METHOD SuperMode : BOOL
VAR_INPUT
END_VAR
IF (*InSync()=TRUE AND *) SyncVertSuperJogExecute_VI AND SuperJogMode_VI THEN
	//jogs are canceled in 'ClearpathLinPPR' FB when SuperJogExecute is set to 0.
	Vert_A.SuperJogExecute_VI :=1;
	Vert_B.SuperJogExecute_VI :=1;
ELSE
	IF JogSeparate_VI = 0 THEN
		Vert_A.SuperJogExecute_VI :=0;
		Vert_B.SuperJogExecute_VI :=0;
	END_IF
END_IF

IF SuperJogMode_VI AND SyncVertSuperJogExecute_VI =0 THEN 	//sync move has to be off to move an individual
	//Vert_A.SuperJogExecute_VI :=VertASuperJog_VI;
	//Vert_B.SuperJogExecute_VI :=VertBSuperJog_VI;

END_IF
END_METHOD

METHOD SyncClampAbsLin : BOOL
VAR_INPUT
END_VAR
IF Clamp_A.Out.InPosition AND Clamp_B.Out.InPosition THEN
	ClampInPosition_PO :=1;
	ELSE ClampInPosition_PO :=0;
END_IF
IF Clamp_A.Out.InTargetPosition AND Clamp_B.Out.InTargetPosition THEN
	ClampInTargetPos_PO :=1;
	else ClampInTargetPos_PO :=0;
END_IF
IF Clamp_A.Out.InMPos AND Clamp_B.Out.InMPos THEN
	ClampIn_M_Pos_PO:=1;
	else ClampIn_M_Pos_PO:=0;
END_IF
CASE SyncClampCase OF
	0: //Ready for move
		IF InSync()=TRUE THEN
			IF Clamp_A.Out.ReadyForMove_PO AND Clamp_B.Out.ReadyForMove_PO THEN
				ClampReadyForMove_PO := TRUE;
				ELSE
					//Msg A or B not readyto move
				END_IF
			ELSE //msg not insync cant move
		END_IF
		IF ClampReadyForMove_PO AND ClampInPosition_PO THEN
			//set request and await execute
			IF bMoveClamp_PI THEN
				Clamp_A.DistancePosReq_PI := ClampDisReq_PI;
				Clamp_B.DistancePosReq_PI := ClampDisReq_PI;
				Clamp_A.bMove_PI :=1;
				Clamp_B.bMove_PI :=1;
				SyncClampCase :=10;
			END_IF
		END_IF
	10: //monitor insync
		bMoveClamp_PI :=0;
		ClampReadyForMove_PO :=FALSE; //step thru case before being able to send again
		IF InSync()=FALSE THEN
			Clamp_A.CancelMove();
			Clamp_B.CancelMove();
			//msg not insync
			SyncClampCase :=90; //syncerror
		END_IF
		//COnfirm Position
		IF ClampInTargetPos_PO THEN
			SyncClampCase:=20;
			ELSE //waiting for move to finish
		END_IF
	20: //Set Ready to Move
		IF InSync()=TRUE THEN
			IF Clamp_A.Out.ReadyForMove_PO AND Clamp_B.Out.ReadyForMove_PO THEN
				ClampReadyForMove_PO := TRUE;
				ELSE
					//Msg A or B not readyto move
				END_IF
			ELSE //msg not insync cant move
		END_IF
		IF ClampReadyForMove_PO THEN SyncClampCase := 0; END_IF
	90: //SyncError
		SyncClampMsg_VO := 'Not in sync abs move was canceld, reset req';
	
END_CASE
END_METHOD

METHOD SyncRotABS : BOOL
VAR_INPUT
END_VAR
IF Rot_A.Out.InPosition AND (Rot_B.Out.InPosition or bFollowerIdleDisengage) THEN
	RotInPosition_PO :=1;
	ELSE RotInPosition_PO :=0;
END_IF
IF Rot_A.Out.InTargetPosition AND (Rot_B.Out.InTargetPosition OR bFollowerIdleDisengage) THEN
	RotInTargetPos_PO :=1;
	ELSE RotInTargetPos_PO :=0;
END_IF
IF Rot_A.Out.InMPos AND Rot_B.Out.InMPos THEN
	RotIn_M_Pos_PO:=1;
	Else RotIn_M_Pos_PO:=0;
END_IF
CASE SyncRotCase OF
	0: //Ready for move
		IF InSync()=TRUE THEN
			IF Rot_A.Out.ReadyForMove_PO AND (Rot_B.Out.ReadyForMove_PO OR bFollowerIdleDisengage) THEN
				RotReadyForMove_PO := TRUE;
				ELSE
					//Msg A or B not readyto move
				END_IF
			ELSE //msg not insync cant move
		END_IF
		IF RotReadyForMove_PO AND RotInPosition_PO THEN
			//set request and await execute
			IF bMoveRot_PI THEN
				Rot_A.DistancePosReq_PI := RotDegReq_PI;
				Rot_B.DistancePosReq_PI := RotDegReq_PI;
				Rot_A.bMove_PI :=1;
				Rot_B.bMove_PI :=1;
				SyncRotCase :=10;
			END_IF
		END_IF
	10: //monitor insync
		bMoveRot_PI :=0;
		RotReadyForMove_PO :=FALSE;	//step thru case before being able to send again
		IF InSync()=FALSE THEN
			Rot_A.CancelMove();
			Rot_B.CancelMove();
			//msg not insync
			SyncRotCase :=90; //syncerror
		END_IF
		//COnfirm Position
		IF RotInTargetPos_PO  THEN
			SyncRotCase:=20;
			ELSE //waiting for move to finish
		END_IF
	20: //Set Ready to Move
		IF InSync()=TRUE THEN
			IF Rot_A.Out.ReadyForMove_PO AND (Rot_B.Out.ReadyForMove_PO or bFollowerIdleDisengage) THEN
				RotReadyForMove_PO := TRUE;
				ELSE
					//Msg A or B not readyto move
				END_IF
			ELSE //msg not insync cant move
		END_IF
		IF RotReadyForMove_PO THEN SyncRotCase := 0; END_IF
	90: //SyncError
		SyncRotMsg_VO := 'Not in sync abs move was canceld, reset req';
	
END_CASE
END_METHOD

METHOD SyncRotJog : BOOL
VAR_INPUT
END_VAR

IF JogSeparate_VI = FALSE THEN
	IF SyncRotJogExecute_VI THEN //JOSEPHBARTONCHANGE IF InSync()=TRUE AND SyncRotJogExecute_VI THEN
		JogRotAExecute_VI :=1;
		JogRotBExecute_VI :=1;
	ELSE
		JogRotAExecute_VI :=0;
		JogRotBExecute_VI :=0;
	END_IF
	ELSE
		//use the jog a or b vi to move items
	
END_IF
END_METHOD

METHOD PUBLIC SyncVertAbsLin : BOOL
VAR_INPUT
END_VAR
IF Vert_A.Out.InPosition AND Vert_B.Out.InPosition THEN
	VertInPosition_PO :=1;
	else VertInPosition_PO :=0;
END_IF
IF Vert_A.Out.InTargetPosition AND Vert_B.Out.InTargetPosition THEN
	VertInTargetPos_PO :=1;
	ELSE VertInTargetPos_PO :=0;
END_IF
IF Vert_A.Out.InMPos AND Vert_B.Out.InMPos THEN
	VertIn_M_Pos_PO :=1;
	ELSE VertIn_M_Pos_PO:=0;
END_IF
CASE SyncVertCase OF
	0: //Ready for move
		IF InSync()=TRUE THEN
			IF Vert_A.Out.ReadyForMove_PO AND Vert_B.Out.ReadyForMove_PO THEN
				VertReadyForMove_PO := TRUE;
				ELSE
					//Msg A or B not readyto move
				END_IF
			ELSE //msg not insync cant move
		END_IF
		IF VertReadyForMove_PO AND VertInPosition_PO THEN
			//set request and await execute
			IF bMoveVert_PI THEN
				Vert_A.DistancePosReq_PI := VertDisReq_PI;
				Vert_B.DistancePosReq_PI := VertDisReq_PI;
				Vert_A.bMove_PI :=1;
				Vert_B.bMove_PI :=1;
				SyncVertCase :=10;
			END_IF
		END_IF
	10: //monitor insync
		bMoveVert_PI :=0;
		VertReadyForMove_PO :=FALSE; //step thru case before being able to send again
		IF InSync()=FALSE THEN
			Vert_A.CancelMove();
			Vert_B.CancelMove();
			//msg not insync
			SyncVertCase :=90; //syncerror
		END_IF
		//Confirm Position
		IF VertInTargetPos_PO THEN
			SyncVertCase:=20;
			ELSE //waiting for move to finish
		END_IF
	20: //Set Ready to Move
		IF InSync()=TRUE THEN
			IF Vert_A.Out.ReadyForMove_PO AND Vert_B.Out.ReadyForMove_PO THEN
				VertReadyForMove_PO := TRUE;
				ELSE
					//Msg A or B not readyto move
				END_IF
			ELSE //msg not insync cant move
		END_IF
		IF VertReadyForMove_PO THEN SyncVertCase := 0; END_IF
	90: //SyncError
		SyncVertMsg_VO := 'Not in sync abs move was canceld, reset req';
	
END_CASE
END_METHOD

METHOD PRIVATE SyncVertJog : BOOL
VAR_INPUT
END_VAR

IF JogSeparate_VI = FALSE THEN
	IF SyncVertJogExecute_VI THEN //IF InSync()=TRUE AND SyncVertJogExecute_VI THEN
		JogVertAExecute_VI :=1;	//JOSEPHBARTONCHANGE1-27-2023 Removed checking in Clamp and Rotary are in synch for vert movement.
		JogVertBExecute_VI :=1;
	ELSE
		JogVertAExecute_VI :=0;
		JogVertBExecute_VI :=0;
	END_IF
	IF InSync()=TRUE AND SyncClampJogExecute_VI THEN
		JogClampAExecute_VI :=1;
		JogClampBExecute_VI :=1;
	ELSE
		JogClampAExecute_VI :=0;
		JogClampBExecute_VI :=0;
	END_IF
	ELSE
		
	//use the jog a or b vi to move items
END_IF
END_METHOD

END_FUNCTION_BLOCK

// ---- Machine System/FBs/CP/ClearpathPositionABS.TcPOU
FUNCTION_BLOCK ClearpathPositionABS //please check comments inside FB to determine clearpath settings before use
VAR_INPUT
	
	//PI (Program Inputs)
		bHomeStart_PI				: BOOL;		//begin Homing sequence
		PowerOn_PI					: BOOL;		//enable motor command from program
		Stop_PI						: BOOL;		//stop command from program
		DistancePosReq_PI			: REAL;		//distanct position request from the program (input in absolute position and valid after homing)
		ManualMove_PI				: BOOL;		//Call manual move method if true
		Mode_PI						: INT;		//0:noMode, 1:Auto, 2:Manual
		bMove_PI					: BOOL;		//begin absolute move 
		VEReq						: LREAL;
		bAltSpeedControl			: BOOL;		//JOSEPHBARTONCHANGE3-28-2023 This allows for outside control of using altspeed
		bPresetMoveTrigger			: BOOL;		//JOSEPHBARTONCHANGE3-28-2023 This allows for tracking when it is a preset position move
		bStopMove			: BOOL;     // Controls the StopMove()
	//VI (visualization input/hmi input)
		HomeReq_VI			: BOOL; 	// Homing sequence
		Reset_VI			: BOOL;		//reset button		
		DisReq_VI			: REAL;		//Disreq for absolute auto move
		JogExecute_VI		: BOOL;		//Call manual move method if true
		SuperJogExecute_VI	: BOOL;		//call super manual move method if true
		SuperJogMode_VI		: bool;		//Super Mode on if true (changes Jog method) use for overtravel or not homed be Cautious
		JogSlow_VI			: BOOL;		//slow manual move
		CW_VI				: BOOL;		//Set Direction for requested move (does not apply to absolute move) True = Clockwise
	//CI (configuration input)
		IN							: CpABS_CI;
		
		EnableOut_FO 		AT %Q* 	: BOOL; 	//enables the clearpath motor
END_VAR
VAR_OUTPUT
	// Outputs
		Out						: CpABS_Out;
		StopCase				: INT; 		//case tracket StopMove()
END_VAR
VAR
	bSimHigh			: BOOL; 	// Simulated High switch for the Rotation axis
	bSimLow				: BOOL; 	// Simulated High switch for the Rotation axis
	AltSpeedCase		: INT;		//case tracker altspeed()
	AltSpeedReq			: BOOL;		//turn altspeed method on
	ResetCase			: int;		//makes a reset instead of an alt speed request (delays the turning off of reset)
	HomeCase			: INT;		//case tracker home()
	JogCase				: INT;		//case tracker Jog()
	SuperJogCase		: INT;		//case tracker SuperJog()
	DisToGoCase			: INT;		//case tracker MoveABSLin() for pulse train que
	PositionCase		: INT;		//case tracker for tracking inposition
	bMoveTrig			: r_trig;	//rtrig for abs move command [used in CNC MDI]
	
	JogReset			: bool;		//used for auto jog reset [stops alt speed from triggering while clearing pulses instead of a full reset]
	SWLimitStatus		: BOOL;		//Used to check if currently within software limits
	error				: INT;		//5: increment error
	PulsesEnabled		: BOOL;		//enable absolute move method to command pulses
	busy				: BOOL;		//move in progress
	MoveComplete		: BOOL;		//all ppr accounted for after move command
	PulseCount			: INT;		//current Pulse Count
	QuePulseDistance	: REAL;		//Distance expected from current pulse train
	expectedPulse		: INT;		//expected pulses from commanded movements at set PPR
	HomeTrig			: R_trig;	//trigger position capture when homing ends
	ATrig				: R_trig;	//counter/trigger to track how many increments of a output have been commanded
	pulseCounter		: r_trig;
	JogRTrig			: R_Trig;	//jog execute trigger
	JogFTrig			: F_Trig;	//Jog Cancel Trigger
	RotRiseLimSwitch		: R_TRIG;	// Rising trigger for rotation limit switch Normally Closed
	RotFallLimSwitch		: F_TRIG;	// Falling trigger for rotation limit switch Normally Open
	ASG					: BOOL;		//all systems go clearpath (if using asg)
	Cancelled			: BOOL;		//move was cancelled requires reset
	CW					: BOOL; 	//direction of motor rotation: CW is true;  CCW is false;
	DistanceToGo		: REAL;		//difference in distance from current position and requested position.  used to determine linear direction
	LastABSEncoder		: DINT;		//last know encoder track to be used for moving status
	isConfigured		: BOOL;		//turns on or off the configuration settings method so it only runs on first scan
	DistPerMRev 		: INT;
	DisPerPulse			: INT;		//distance per pulse based on configuration inputs
	PulsesToSend		: INT;		//Pulses to send for Absolute move
	CWABS				: Bool;		//Direction for abs Move [Check against pulse wrong dir]
	PulseQueSet			: BOOL;		//start pulses for move
	LastDistanceposReq	: REAL;		//last abs move request (keeps track of InTargetPosition)
	ABSHiLimit	: DINT;
	ABSLoLimit 	: Dint;
	//FI (Field Inputs)

	HLFB_FI	 		AT %I*	: BOOL;		// high level feedback sensors
	bInputBCom_FI	AT %I*	: BOOL;		// check sum for inputb signal	(double check that direction is actually signaled to motor)
	ABSEncoder_FI	AT %I*	: DINT;		//absoulte multiturn encoder
	
	//Linear Homing Variables
	bHigh_FI		AT %I*	: BOOL;
	bLow_FI			AT %I*	: BOOL;
	bHome_FI		AT %I*	: BOOL;
	
	bTest : BOOL;
	
	//FO (Field Outputs)
	HLFB24V_FO 			AT %Q*	: BOOL :=1;	//high level feedback 24v power if needed to used el2008 //default set to true so that hlfb is fucntional
	InputAOut_FO 		AT %Q* 	: BOOL; 	//input A of clearpath motor, output from plc
	InputBOut_FO 		AT %Q* 	: BOOL; 	//input B of clearpath motor, output from plc
END_VAR
VAR RETAIN 
	
	
END_VAR

VAR_IN_OUT

END_VAR

(* Check clearpath settings before use*)
	(* Check the input filter setting for inputA and inputB.   Also check PPR setting, CntsPerPulse, HLFBsetting, and The type of axis,  
		Place clearpath in correct mode of operation Mode for this FB is position 
		Check what Homing setting is used on the clearpath motor	
		check to make sure that the resolution of movement commands matches gearbox compatibiltiy, and plc scan compatability
		
		How the FB works Details:
			1st scan sets configuration using MechDrive_CI()
			Each scan CP motor direction is set based off CW variable
			LocatePosition() drives limit switches and rotary cam limit quadrants
			Pulses are counted using ppr() to move with hlfb rising trig counter.  Expected pulses are tracked with inputA_FO rising trig
			Enable checks for enable signal, cancelled state, and stop_PI state before turning on motor or disenable
			reset: cp motors require an enable off to reset after ac loss...ie estop w/contactor.  it also resets cancelled bit and busy bit (requires reset_vi to run)
			
			Moves are called using homing sequence, Absolute movement, or with manual movement and all require homing.
			after homing absolute movement within software limit_CI is available or manual jog.  Manual jog is set to single pulse method by default
			After Homing Position is tracked using 'DistancePos_PO'
			ABsolute move chains clearpath pulses together to create a smooth motion profile. 
				Pulses sent are tracked against 'DistancePosReq_PI' and 'DistancePos_PO'  When expected pulses are within range of requested position then 'pulsecount' is reset
	*)
(*configruation input setting*)
IF isConfigured = 0 THEN MechDrive_CI(); bHigh_FI := TRUE; END_IF	//run once to set configuration on init

//Handle alternate speed
AltSpeedReq := bAltSpeedControl OR AltSpeedReq;
//Pin outs Clockwise (CW) or Counter Clockwise (CCW)
IF CW THEN	InputBOut_FO := 1;	ELSE InputBOut_FO := 0; 	END_IF //sets direction of movement at motor - check this (add bcom direction pin check)
LocatePosition();				//rotary position of the cam wheel  //also includes a double sensor check for SensorCheck_PO  //Also locates position for linear system for limit sensors //Limits
//Triggers
	//pulseCounter(clk:=HLFB_FI);		//high Level feedback counter based off direction (replaced by abs encoder)
	HomeTrig(clk:=Out.Homed_PO);		//used in ppr() to set pulses to zero after homing
	ATrig (clk:=InputAOut_FO);		//counts pulses sent to motor (clearpath should move based on InputA Rising Trig (check settings in CP to be sure - options are for rising or falling trig)
	JogRTrig(CLK:=JogExecute_VI,);	//Starts Jog()
	JogFTrig(CLK:=JogExecute_VI,);	//Cancels Jog() movement
	bMoveTrig(Clk:=bmove_PI,); 		//confirms that move has triggered and then can check MDI MCode Req Pos	
IF Mode_PI = 2 THEN	
	IF SuperJogMode_VI = 0 THEN
		Jog();
	ELSE
		SuperJog();
	END_IF
	out.ModeMsg_VO := 'Manual Mode engaged';
END_IF
IF Mode_PI = 1 THEN
	out.ModeMsg_VO := 'Auto Mode Engaged';
	DistancePosReq_PI:=DisReq_VI;
	MoveAbsLin();
END_IF
	ABSEncoder();			//tracking of the abs encoder against inputB pulses (default for most use cases) use ppr if using the pulse signals from clearpath
	Home();

//moved movedone into movement manual call and abs move call
MoveDone();						//check if movement is complete (will either check pulses against expected pulses or will check for asg
Enable();						//check for motor enable status and try to enable the motor if PowerOn_PI is true
Reset();						//if reset button turn power off, reset cancelled, and reset busy
IF stop_PI THEN CancelMove(); END_IF	//This requires a reset afterwards to move again
IF GVL_HMI.AutoMode THEN StopMove(); END_IF // Must call axis auto stopping every cycle.

METHOD ABSEncoder : BOOL
VAR_INPUT
END_VAR
VAR
	bTest : BOOL;
END_VAR
//pulsecount is now turned into absolute encoder
//will need to check pulsecount math against encoder and confirm rounding does not cause fb and motor to hunt between pulses
Out.DistancePos_PO :=  (ABSEncoder_FI-in.ABSEncoderZero_CI)/in.ABSEncoderScaler_CI;

ABSHiLimit:= (IN.ABSEncoderZero_CI + (In.ABSEncoderScaler_CI*(In.SWLimit_Hi_CI+5))); //JosephBartonChange1-11-2023 THISISIT ABSEncoderZero_CI
ABSLoLimit:= (In.ABSEncoderZero_CI + (IN.ABSEncoderScaler_CI*(In.SWLimit_Lo_CI-5))); //JosephBartonChange1-11-2023
IF ATrig.Q AND Cancelled = 0 THEN //pulse sent counter rtrg
	IF InputBOut_FO = 1 THEN 
		//QuePulseDistance := QuePulseDistance + In.DisPerPulse_CI; //does not account for cnt per rev yet
		PulsesToSend := PulsesToSend-1; //Track ABS Pulses sent  [went pos dir so remove one from que]
		ELSE 
			//QuePulseDistance := QuePulseDistance - In.DisPerPulse_CI;
			PulsesToSend := PulsesToSend+1; //Track ABS Pulses sent  [went neg dir so add one from que]
	END_IF
	//disperpulse_CI must be calibrated on axis and set in settings
END_IF

IF Cancelled = 1 THEN
	//expectedPulse := pulsecount; 			//removed expectedpulse in favor of QuePulseDistance with the abs encoder Ref the linppr if editing
	//QuePulseDistance := 0;
	Out.ExpDistancePos_PO := Out.DistancePos_PO;
END_IF
IF  movecomplete = 1 THEN //ppr mode
	 //Out.ExpDistancePos_PO := PulseCount/2;
	 Out.ExpDistancePos_PO := Out.DistancePos_PO;
	 //QuePulseDistance:=0;
END_IF
IF  PowerOn_PI =0 THEN
	 Out.ExpDistancePos_PO := Out.DistancePos_PO;
	 //QuePulseDistance:=0;
END_IF
Out.DistancePos_PO := Out.DistancePos_PO; //change distancePOs_PO to float if needed
END_METHOD

METHOD PUBLIC AltSpeed : BOOL
VAR_INPUT
END_VAR
(*clearpath requires at least a 20ms delay where the enable signal is pulsed off to realize alternate speed *)

//start
CASE AltSpeedCase OF
	0:
		IF FIND(STR1:='VERT', STR2:=IN.MotorName) = 0 THEN
			altspeedcase := 10;
		ELSE
			altspeedcase := 100;
		END_IF
	10:
		EnableOut_FO := 1;
		AltSpeedCase := 20;
	20:
		EnableOut_FO := 1;
		AltSpeedCase := 30;
	30:
		EnableOut_FO := 0;
		AltSpeedCase := 40;
	40:
		EnableOut_FO := 0;
		AltSpeedCase := 50;
	50:
		EnableOut_FO := 0;
		AltSpeedCase := 60;
	60:	
		EnableOut_FO := 1;
		//Look for 'AltSpeedCase' to be set to '0' in the call function
	
	90: //error or message
	
	100: 
		EnableOut_FO := 1;
		AltSpeedCase := 110;
	110:
		EnableOut_FO := 1;
		AltSpeedCase := 120;
	120:
		EnableOut_FO := 1;
		AltSpeedCase := 130;
	130:
		EnableOut_FO := 0;
		AltSpeedCase := 140;
	140:
		EnableOut_FO := 0;
		AltSpeedCase := 150;
	150:
		EnableOut_FO := 0;
		AltSpeedCase := 200;
	200: 
		EnableOut_FO := 1;
		AltSpeedCase := 110;
	210:
		EnableOut_FO := 1;
		AltSpeedCase := 220;
	220:
		EnableOut_FO := 1;
		AltSpeedCase := 230;
	230:
		EnableOut_FO := 0;
		AltSpeedCase := 240;
	240:
		EnableOut_FO := 0;
		AltSpeedCase := 250;
	250:
		EnableOut_FO := 0;
		AltSpeedCase := 60;
END_CASE
END_METHOD

METHOD PUBLIC CancelMove : BOOL
VAR_INPUT
END_VAR

VAR
	rCanceledEncoderValue : REAL;
END_VAR
EnableOut_FO 	:= 0;		//only way to clear out overstacked increment calls is to turn enable off and then on
//PowerOn_PI		:=0;	//turn off power on [this is a program input and can't be turned off here] check this to see if still needed[was affecting homecase]
Cancelled	:=1;	//cancelled move needs to be reset
Out.ExpDistancePos_PO := Out.DistancePos_PO; //change distancePOs_PO to float if needed
DistancePosReq_PI:=Out.DistancePos_PO;	// get rid of any requestd move during cancel (must recall it after cancel)
DisToGoCase :=0;
PulsesToSend :=0;
//MCODE Flag
AltSpeedReq :=0;	//clear alt speed mode	
AltSpeedCase :=0;	
InputAOut_FO :=0;
// message (move was canceled)
Out.Error4Msg_VO := 'Cancelled, reset to move motor';
END_METHOD

METHOD PUBLIC Enable : BOOL 	//attempts to enable the motor based on stop_PI, Cancelled, and PowerOn_PI
VAR_INPUT
END_VAR
IF Stop_PI =0 AND cancelled =0 AND PowerOn_PI =1 and ResetCase=0 THEN
	EnableOut_FO :=1;
	IF altSpeedReq THEN
		AltSpeed();				//calls altspeed to cycle thru if homing or manual mode requests a slower mode
	END_IF
ELSE 
	EnableOut_FO :=0;	//message to say stop is on (check this)
END_IF


//power on

//check if asg
IF EnableOut_FO =1 AND HLFB_FI =0 THEN
	Out.ErrorMsg_VO := 'Servo enabled but HLFB not on';
END_IF

//if no asg power off and repeat
END_METHOD

METHOD PUBLIC Error : BOOL
VAR_INPUT
END_VAR
// if hlfb pulses do not move in set timeframe after movement call then call error for motor
END_METHOD

METHOD PUBLIC Home : BOOL
VAR_INPUT
END_VAR
//If encoder field is within the CI limits then machine counts as homed.  If homing seq is needed to check slippage periodically it can be added in this method
IF ABSEncoder_FI >= ABSLoLimit AND ABSEncoder_FI <= ABSHiLimit THEN
	out.Homed_PO := 1;
	Out.HomeMsg_VO := 'Axis is within home limits';
	ELSE
		Out.Homed_PO :=0;
		Out.HomeMsg_VO := 'Axis not within home limits check overtravel';
END_IF

//MAIN HOMING SEQUENCE

CASE HomeCase OF 
	0:	//Main home Sequence [Also stops movement]
		
		
		IF HomeReq_VI  THEN	
			IF IN.Limit_NC_NO_CI = 0 THEN	//NC limit switch configuration
				IF bLow_FI THEN //set direction via hmi unless on a limit switch then default to locateposition()
					CW := 0;
					SendPulse();
				ELSE
					CancelMove();
					//in.ABSEncoderZero_CI := ABSEncoder_FI;
					HomeCase :=10;
				END_IF
			ELSE	//NO limit switch configuration
				IF NOT(bLow_FI) THEN //set direction via hmi unless on a limit switch then default to locateposition()
					CW := 0;
					SendPulse();
				ELSE
					CancelMove();
					HomeCase :=10;
				END_IF
			END_IF
			
		ELSE
			IF	Reset_VI  OR Stop_PI THEN		
				CancelMove();
				HomeCase :=10;
			END_IF
		END_IF
	10:	//go for auto jog reset
		IF cancelled THEN HomeCase :=20; END_IF
		
	20: //auto Reset cycle
		IF InLimits(Out.DistancePos_PO) THEN HomeCase :=30; ELSE HomeCase:=95;  END_IF
	30: HomeCase :=31; //10 scan delay
	31: HomeCase :=32;
	32:	HomeCase :=33;
	33: HomeCase :=34;
	34: HomeCase :=35;
	35: HomeCase :=36;
	36: HomeCase :=37;
	37: HomeCase := 38;
	38: HomeCase := 39;
	39: HomeCase :=40;
	40: //send reset
		JogReset := 1;
		HomeCase :=50;
	50: //wait for reset
		IF JogReset=0 THEN HomeCase :=90; END_IF 
	60:
	70:
	80:
	90: IF HomeReq_VI =TRUE THEN HomeCase :=0; END_IF
	95: //outside of limits
		IF Reset_VI THEN HomeCase:=90; END_IF //no autoreset if outside limits
END_CASE
//slippage Test Periodically if desired

//limit switch and home switch configuration
	(*IF IN.HomingSet_CI = 2 THEN //homing sensor not used - home to low sensor
	bHome_FI := bLow_FI; 
	//message homing sensor not used
	END_IF
	
	IF IN.HomingSet_CI = 3 THEN //homing sensor not used - home to Hi sensor
		bHome_FI := bHigh_FI; 
		//message homing sensor not used
	END_IF
	//error catch for if InputBout wire fails and ends up homing unknown direction repeatedly
	IF PowerOn_PI = 0 THEN HomeCase :=0; END_IF
	IF Stop_PI = 1 THEN HomeCase := 0; END_IF
	//check the InputBOut com using EL1008 input channel to determine that the pulse did work
	//message
	IF bhomestart_PI = 1 THEN HomeCase :=0; AltSpeedReq := 1; AltSpeedCase:=0; END_IF
	CASE HomeCase OF
		0://set pulses equal so that movement can begin and check direction
			IF bHomeStart_PI =1 AND Stop_PI = 0  THEN
				HomeCase := 10;
				bhomeStart_PI :=0;
				AltSpeedReq := 1;				//set slow mode and alternate speed in clearpath
				//AltSpeedCase := 0;			//may need this to start slow speed
				//ExpectedPulse := PulseCount;	//Make movement available no matter the pulse count discrepancy
				Out.ExpDistancePos_PO := Out.DistancePos_PO;
				InputAOut_FO :=0;
				Out.Homed_PO :=0;
			END_IF
		(*5:	
			IF Stop_PI = 0  THEN
				HomeCase := 10;
				bhomeStart_PI :=0;
				AltSpeedReq := 1;				//set slow mode and alternate speed in clearpath
				AltSpeedCase := 0;
				ExpectedPulse := PulseCount;	//Make movement available no matter the pulse count discrepancy
				Homed_PO :=0;
			END_IF*)
			
		10:// homing sequence
			IF  Stop_PI = 0  THEN
				Out.Homed_PO :=0;
				//check this: reseting expected to match pulse count so that homeing will start if there is a mismatch
				//decide homing direction and homing method //make flag large enough to hit home switch and the limit switch
				IF IN.Limit_NC_NO_CI =0 THEN	//NC switch configuration
					IF bHigh_FI =1 AND bLow_FI =1 THEN	//using normally closed sensor (flag is not on either limit switch)
						IF IN.HomingSet_CI =2 THEN cw := 0; ELSIF IN.HomingSet_CI =3 THEN cw :=1; END_IF //go to high or low first if no limit switch tripped
					END_IF
				ELSE	//NO switch Configuration
					IF bHigh_FI =0 AND bLow_FI =0 THEN	//using normally closed sensor (flag is not on either limit switch)
						IF IN.HomingSet_CI =2 THEN cw := 0; ELSIF IN.HomingSet_CI =3 THEN cw :=1; END_IF //go to high or low first if no limit switch tripped
					END_IF
				END_IF
				//if inputA is hi then turn off (takes 2 cycles to output an increment at cp motor)
					(*if pulses expected = pulse count then do the next move *)
				IF AltSpeedCase = 60 THEN SendPulse(); END_IF
				IF IN.Limit_NC_NO_CI =0 THEN	//NC switch configuration
					IF bHome_FI =0 THEN //use nc switch for sensor [at home position]
						bHomeStart_PI :=0;
						Cancelmove();
						HomeCase := 20;
					END_IF
					ELSE				//NO switch configuration
					IF bHome_FI =1 THEN //use no switch for sensor [at home position]
					bHomeStart_PI :=0;
					Cancelmove();
					HomeCase := 20;
				END_IF	
				END_IF
				(*check this - add in an extra cycle before setting home that moves away from the 
					homed spot in same direction to confirm trigger positino comes on same side of sensor each time*)
			END_IF
		20:	//extra scan before homed
			HomeCase :=50;	//this scan is required to allow for a cancelled move reset after homing
		
		50://after homing reset motor and cancelled bit
			
				Out.Homed_PO := 1;
				//cancelled :=0;	//resets motor after initial homing
				
				//pulsecount :=0; 
				//expectedPulse :=0;
				Out.DistancePos_PO :=0; //set this to calibrated abs value
				Out.ExpDistancePos_PO :=0; //check this prob need to set to Out.distancepos_po after it calibrates
				testbool := TRUE;
				HomeCase := 0;	//back to the start
		90://reset to default or?
		
	END_CASE *)
END_METHOD

METHOD PUBLIC InLimits : BOOL
VAR_INPUT
	Req	: REAL;	//reqested degree or position from abs move to be evaluated for limits
END_VAR
//only valid after homing
InLimits := TRUE;
IF IN.SWLimit_Hi_CI <=0 OR IN.SWLimit_Lo_CI >0 THEN		//check this (may need to have a neg hi at some point)
	//message to say no limits are set
	Out.Error2Msg_VO := 'No limits are set in CI settings';
	InLimits :=FALSE;	
END_IF
IF Req <= IN.SWLimit_Hi_CI AND Req >= IN.SWLimit_Lo_CI THEN
	InLimits := TRUE;
	ELSE
		InLimits :=FALSE;
		Out.Error2Msg_VO := 'Requested move is outside of software limits';
END_IF
END_METHOD

METHOD PUBLIC Jog : BOOL
VAR_INPUT
END_VAR

//add software limits check this
CASE JogCase OF 
	0:	//Main Jog Sequence [Also stops movement]
		IF JogSlow_VI THEN AltspeedReq :=1; ELSE AltSpeedReq :=0;   END_IF
		
		IF JogExecute_VI AND Out.Homed_PO =1 AND SWLimitStatus=TRUE THEN	//if last move is done then allow for manual increment also required to be at home //check sensor check
			IF IN.Limit_NC_NO_CI = 0 THEN	//NC limit switch configuration
				IF bHigh_FI AND bLow_FI THEN //set direction via hmi unless on a limit switch then default to locateposition()
					IF CW_VI = 1 	THEN	CW := 1; 	ELSE CW:=0; 	END_IF
					IF bhigh_fI = 0	THEN 	CW:=0; 		END_IF
					IF bLow_FI = 0 	THEN 	CW:=1; 		END_IF
				END_IF
			ELSE	//NO limit switch configuration
				IF bHigh_FI =0 AND bLow_FI  = 0 THEN //set direction via hmi unless on a limit switch then default to locateposition()
					IF CW_VI = 1 	THEN	CW := 1; 	ELSE CW:=0; 	END_IF
					IF bhigh_fI = 1	THEN 	CW:=0; 		END_IF
					IF bLow_FI = 1 	THEN 	CW:=1; 		END_IF
				END_IF
			END_IF
			IF AltspeedReq THEN			// slowjog if altspeed is requested and wait for case 60
				IF AltspeedCase = 60 THEN
					SendPulse();
				END_IF
			ELSE
					SendPulse();		//send pulse for reg speed jog
			END_IF
		ELSIF JogExecute_VI THEN
				IF ABSEncoder_FI >= ABSHiLimit OR (IN.Limit_NC_NO_CI = 0 AND bHigh_FI =0) OR (IN.Limit_NC_NO_CI = 1 AND bHigh_FI =1)THEN
					CW := 0;
					SendPulse();		//send pulse for reg speed jog
				ELSIF ABSEncoder_FI <= ABSLoLimit OR (IN.Limit_NC_NO_CI = 0 AND bLow_FI =0) OR (IN.Limit_NC_NO_CI = 1 AND bLow_FI =1) THEN
					CW := 1;					
					SendPulse();		//send pulse for reg speed jog
				END_IF
		ELSE
			IF	JogExecute_VI  = FALSE THEN		
				CancelMove();
				JogCase :=10;
			END_IF
		END_IF
	10:	//go for auto jog reset
		IF cancelled THEN jogCase :=30; END_IF
		
	20: //auto Reset cycle
		IF InLimits(Out.DistancePos_PO) THEN JogCase :=30; ELSE JogCase:=95;  END_IF
	30: JogCase :=31; //10 scan delay
	31: JogCase :=32;
	32:	JogCase :=33;
	33: JogCase :=34;
	34: JogCase :=35;
	35: JogCase :=36;
	36: JogCase :=37;
	37: JogCase := 38;
	38: JogCase := 39;
	39: JogCase :=40;
	40: //send auto jog reset
		JogReset := 1;
		JogCase :=50;
	50: //wait for jog to reset
		IF JogReset=0 THEN JogCase :=90; END_IF 
	60:
	70:
	80:
	90: IF JogExecute_VI =TRUE THEN JogCase :=0; END_IF
	95: //outside of limits
		if Reset_VI then JogCase:=90; End_if //no autoreset if outside limits
	
END_CASE
END_METHOD

METHOD PUBLIC LocatePosition : Bool //determines if sensorcheck is on and working.  Enables movement
VAR_INPUT
END_VAR
	// Setup the switches for rotational axis.
IF IN.bIsRotationAxis THEN
	RotRiseLimSwitch(CLK := bHigh_FI);
	RotFallLimSwitch(CLK := bHigh_FI);
	IF IN.Limit_NC_NO_CI = 0 THEN
		IF RotRiseLimSwitch.Q THEN
			bSimHigh := TRUE;
			bSimLow  := TRUE;
		END_IF
		IF RotFallLimSwitch.Q THEN
			IF CW_VI THEN
				bSimHigh := FALSE;
				bSimLow  := TRUE;
			ELSE
				bSimHigh := TRUE;
				bSimLow  := FALSE;
			END_IF
		END_IF
	ELSE
		IF RotRiseLimSwitch.Q THEN
			bSimHigh := FALSE;
			bSimLow  := FALSE;
		END_IF
		IF RotFallLimSwitch.Q THEN
			IF CW_VI THEN
				bSimHigh := TRUE;
				bSimLow  := FALSE;
			ELSE
				bSimHigh := FALSE;
				bSimLow  := TRUE;
			END_IF
		END_IF
	END_IF
	
	bHigh_FI := bSimHigh;
	bLow_FI  := bSimLow;
END_IF


// Linear axis limit sensors
(*		bHigh_FI		AT %I*	: 	BOOL;
		bLow_FI			AT %I*	: 	BOOL;
		bHome_FI		AT %I*	: 	BOOL;*)
//NC limit sensor configuration
IF IN.Limit_NC_NO_CI = 0 THEN	
	IF bHigh_FI =0 AND bInputBCom_FI =1 AND CW = 1 THEN	//use normally closed sensor and check inputb(-) [applies when trying to move past limit]
		cancelmove();
		CW := 0;	//require next move to be in Neg direction or CCW  //manual move will need to be used to get off limit switch check this
		//message saying that high limit as been exceeded or inputbcom is not connected
		Out.ErrorMsg_VO := 'High Limit reached, reset and move away from limit';
	END_IF
	IF bLow_FI =0 AND bInputBCom_FI = 0 AND CW =0 THEN	//use normally closed sensor and check inputb(-) [applies when trying to move past limit]
		cancelmove();
		CW :=1;	//require next move to be in Neg direction or CCW //manual move will need to be used to get off limit switch check this
		//message saying that Low limit as been exceeded or inputbcom is not connected
		Out.ErrorMsg_VO := 'Low Limit reached, reset and move away from limit';
	END_IF
	//check for abs encoder slip
	IF bHigh_Fi = 0 THEN
		IF ABS(ABSEncoder_FI - ABSHiLimit)> 100 THEN
			Out.Error3Msg_VO := 'Encoder descrepancy at high limit, please confirm no slippage has occured.  Reset encoder calibration in CI settings if needed.';
		END_IF
	END_IF
	IF bLow_FI = 0 THEN
		IF ABS(ABSEncoder_FI - ABSLoLimit)> 100 THEN
			Out.Error3Msg_VO := 'Encoder descrepancy at low limit, please confirm no slippage has occured.  Reset encoder calibration in CI settings if needed.';
		END_IF
	END_IF
ELSE
	//NO limit sensor configuration
	//additional option to use a N/O sensor if desired....not suggested
	IF bHigh_FI =1 AND bInputBCom_FI =1 AND CW = 1 THEN	//use normally closed sensor and check inputb(-) [applies when trying to move past limit]
		cancelmove();
		CW := 0;	//require next move to be in Neg direction or CCW  //manual move will need to be used to get off limit switch check this
		//message saying that high limit as been exceeded or inputbcom is not connected
		Out.ErrorMsg_VO := 'High Limit reached, reset and move away from limit';
	END_IF
	IF bLow_FI =1 AND bInputBCom_FI = 0 AND CW =0 THEN	//use normally closed sensor and check inputb(-) [applies when trying to move past limit]
		cancelmove();
		CW :=1;	//require next move to be in Neg direction or CCW //manual move will need to be used to get off limit switch check this
		//message saying that Low limit as been exceeded or inputbcom is not connected
		Out.ErrorMsg_VO := 'Low Limit reached, reset and move away from limit';
	END_IF
	//check for abs encoder slip
	IF bHigh_Fi = 1 THEN
		IF ABS(ABSEncoder_FI - ABSHiLimit)> 100 THEN
			Out.Error3Msg_VO := 'Encoder descrepancy at high limit, please confirm no slippage has occured.  Reset encoder calibration in CI settings if needed.';
		END_IF
	END_IF
	IF bLow_FI = 1 THEN
		IF ABS(ABSEncoder_FI - ABSLoLimit)> 100 THEN
			Out.Error3Msg_VO := 'Encoder descrepancy at low limit, please confirm no slippage has occured.  Reset encoder calibration in CI settings if needed.';
		END_IF
	END_IF
END_IF
IF Out.DistancePos_PO <=In.SWLimit_Hi_CI AND Out.DistancePos_PO >= In.SWLimit_Lo_CI THEN
	SWLimitStatus := TRUE;
	OUt.LimitsMsg_VO := '';
	ELSE
		SWLimitStatus :=FALSE;
		OUt.LimitsMsg_VO := 'Not inside Software limits, use super mode to move past overtravel';
		//add in ability to jog off of limit
		IF Out.DistancePos_PO >= In.SWLimit_Hi_CI AND CW=1 THEN
			CancelMove();
			CW :=0;
			OUt.LimitsMsg_VO := 'Low SW limit, reset and use super mode to move past overtravel';
		END_IF
		IF Out.DistancePos_PO <= In.SWLimit_Lo_CI AND CW=0 THEN
			CancelMove();
			CW :=1;
			OUt.LimitsMsg_VO := 'High SW limit, reset and use super mode to move past overtravel';
		END_IF
END_IF
END_METHOD

METHOD PUBLIC MechDrive_CI : BOOL
VAR_INPUT
END_VAR
// 0: motor only(rot), 1: Motor and gear(rot), 2: Motor w/gear and screw(lin), 3: Motor w/screw only(lin), 4: Motor w/gear and pulley(lin),  5: Motor w/pulley(lin), 8: bypass mode
(*		DistPerMRev_CI		:	INT;	//distance traveled per rev		(Calculate your own pitch and lead w/gearbox combo must set MechDriveType_CI to 8 to bypass internal calc)
		DegPerMRev_CI		:	INT;	//distance traveled per rev		(Calculate your own pitch and lead w/gearbox combo must set MechDriveType_CI to 8 to bypass internal calc)
		DisPerFPulley_CI	:	INT;	//distance traveled per rev of final pulley (mm)
		GearRatio_CI		:	INT;	// GearRatio motor to moving part (XX:1) (gearbox and lead included in calc for vert axis) (use this for gearbox and pulleys as well)
		Lead_CI				:	INT;	// Lead of Screw if used (mm)			 (gearbox and lead included in calc for vert axis)	
*)

IF IN.MechDriveType_CI = 2 THEN	//2: Motor w/gear and screw(lin)
	DistPerMRev := IN.Lead_CI/IN.GearRatio_CI;	//driven mech ex 4mm/40 = .1mm per rev
	Out.MechTypeMsg_VO := 'Motor w/gear ratio and screw - no Degrees available [no rotary by default]';
	IF IN.GearRatio_CI <=0 OR IN.Lead_CI <=0 THEN
		isconfigured :=0;
		Out.MechTypeMsg_VO := 'GearRatio_CI or Lead_CI not configured please configure to continue';
	END_IF
END_IF

IF IN.MechDriveType_CI = 3 THEN	//3: Motor w/screw only(lin)
	DistPerMRev := IN.Lead_CI;		//driven mech ex 4mm = 4mm per rev
	Out.MechTypeMsg_VO := 'Motor w/screw - no Degrees available [no rotary by default]';
	IF IN.Lead_CI <=0 THEN
		isconfigured :=0;
		Out.MechTypeMsg_VO := 'Lead_CI not configured please configure to continue';
	END_IF
END_IF

IF IN.MechDriveType_CI = 4 THEN	//4: Motor w/gear and pulley(lin),
	DistPerMRev := IN.DisPerFPulley_CI/IN.GearRatio_CI;	//pulley circumference (20t at10 ~ 200mm per fin rev/gear ratio (40) = 5mm/motor rev
	Out.MechTypeMsg_VO := 'Motor w/gear ratio and pulley [no Degree used by default (linear pulley drive) if a rotary either use bypass or use type 1 and include pulley in gear ratio]';
	IF IN.GearRatio_CI <=0 OR IN.DisPerFPulley_CI <=0 THEN
		isconfigured :=0;
		Out.MechTypeMsg_VO := 'GearRatio_CI or DisPerFPulley_CI not configured please configure to continue';
	END_IF
END_IF

IF IN.MechDriveType_CI = 5 THEN	//5: Motor w/pulley(lin);
	DistPerMRev := IN.DisPerFPulley_CI;	//pulley circumference (20t at10 ~ 200mm per fin rev/gear ratio (40) = 5mm/motor rev
	Out.MechTypeMsg_VO := 'Motor w/pulley [no Degree used by default (linear pulley drive) if a rotary either use bypass or use type 1 and include pulley in gear ratio]';
	IF IN.DisPerFPulley_CI <=0 THEN
		isconfigured :=0;
		Out.MechTypeMsg_VO := 'DisPerFPulley_CI not configured please configure to continue';
	END_IF
END_IF

IF IN.MechDriveType_CI = 8 THEN	//8 mechdrivetype is bypassed and is set via DistPerMRev_CI or DegPerMRev_CI;
	DistPerMRev := IN.DistPerMRev_CI;
	Out.MechTypeMsg_VO := 'MechDriveType is bypassed - use DegPerMRev_CI or DistPerMRev_CI';
	IF IN.DistPerMRev_CI <=0  THEN
		isconfigured :=0;
		Out.MechTypeMsg_VO := 'DistPerMRev_CI not configured please configure to continue';
	END_IF
END_IF

IF IN.InputFilter_CI <=0 THEN
	isconfigured :=0;
	Out.ConfigMSG_VO := 'Input filter not configured, please check InputFilter_CI and clearpath motor settings';
END_IF

//linear axis
DisPerPulse := (DistPerMRev*IN.cntpulseSet_CI/32000);	//check this (Likely not a correct calc)
isConfigured :=1;	//sets configuration to true so that this block only runs once
END_METHOD

METHOD PUBLIC MoveAbsLin : BOOL
VAR_INPUT
END_VAR
IF Out.Homed_PO THEN
	CASE PositionCase OF
		0:
			IF ABS(out.DistancePos_PO-LastDistanceposReq) < In.MoveABSTol_CI THEN 
				Out.InTargetPosition:=1; ELSE Out.InTargetPosition:=0; 
			END_IF
			PositionCase :=10;
		10: PositionCase :=20;
		20: PositionCase :=30;
		30: PositionCase :=40;
		40: PositionCase :=50;
		50: PositionCase :=90;
		90: PositionCase :=0;
	END_CASE
	IF ABS(VEReq - Out.DistancePos_PO) < In.MoveABSTol_CI THEN
		Out.InMPos :=1; ELSE Out.InMPos:=0;
	END_IF
	IF bMoveTrig.Q THEN Out.InMPos :=0; END_IF //Set the MPos to false after move command
	CASE DisToGoCase OF
		0:	//Readyto Take Command
			IF ABS(out.DistancePos_PO-Out.ExpDistancePos_PO) < In.MoveABSTol_CI THEN Out.InPosition:=1; END_IF	//check if current pos is within tolerance
			IF Out.InPosition THEN Out.ReadyForMove_PO :=1; END_IF		//Only ready if in position
			IF Out.ReadyForMove_PO THEN
				IF bMove_PI AND InLimits(DistancePosReq_PI)THEN  //If move is within set limits and called in Prog then execute move
					
					DisToGoCase :=10;
					//set MCode Received Bit [Confirm acted in end case] (this is important for aux axis in cnc VE Variable calls)
				END_IF
			END_IF
		10: //check what quePulseDistance should be and set it
			IF bPresetMoveTrigger THEN
				PulsesToSend := REAL_TO_INT((DistancePosReq_PI - Out.DistancePos_PO) * 1.5); //Gets number of pulses to send When moving to set position.
			ELSE
				PulsesToSend := REAL_TO_INT((DistancePosReq_PI - Out.DistancePos_PO)/In.DisPerPulse_CI); //Gets number of pulses to send
			END_IF
			IF PulsesToSend >0 THEN CWABS:=1; ELSE CWABS:=0; END_IF 	//Sets direction for pulses (pos CW[true] neg CW[False]
			bMove_PI :=0;	//Set Req back to false
			LastDistancePosReq := DistancePosReq_PI; //set for target
			Out.ReadyForMove_PO:=0;	//set busy with abs move
			DisToGoCase :=20;
		20: //set the if homed statement for direction control set that here and move to next case
			IF CWABS THEN CW:=1; ELSE CW:=0; END_IF	//Check abs direction each round of pulse send
			IF ABS(PulsesToSend) >0 THEN 
				PulsesEnabled:=1; 
			ELSE 	
				PulsesEnabled :=0;
				DisToGoCase :=30; //if no more pulses move on to case 30 to check the location toleranceS
					// JOSEPHBARTONCHANGE3-28-2023 Reset bPresetMoveTrigger to FALSE, because the move has ended, so no more preset move.
				IF bPresetMoveTrigger THEN
					bPresetMoveTrigger := FALSE;
				END_IF
				
			END_IF	//if any pos or neg pulses then enable pulses
			Out.InPosition :=0;
			IF PulsesEnabled =1 AND Stop_PI = 0 AND EnableOut_FO =1 AND CW = bInputBCom_FI THEN	//check for the motor being on before incrementing the distancepos from disreq	
				//if inputA is hi then turn off (takes 2 cycles to output an increment at cp motor)
				IF CW = CWABS THEN
					SendPulse();	
				ELSE //Message CW Not equal CWABS
						CancelMove();
						Reset_VI := TRUE;
				END_IF	
			ELSE
				error := 5; //check the inputbcom_FI feedback
			END_IF	
			//if input filter of clearpath is too high sometimes these pulses will not register (needed to maintain ability to chain moves)  Otherwise can use asg and movedone
		30: //count pulses and and when enough pulses set pulses(rounded) not enabled set moving tag
			IF ABS(out.DistancePos_PO-DistancePosReq_PI) < In.MoveABSTol_CI THEN
				Out.InPosition:=1; Out.ABSMoveMsg_VO:='In Position';//Position Reached flag and msg
				DisToGoCase := 40;
				ELSE DisToGoCase :=99; //error
			END_IF
			DisToGoCase :=40;
		40: //add a few scan frames to allow inposition and intarget to be bypassed
			DisToGoCase:=41;
		41:	DisToGoCase:=42;
		42:	DisToGoCase:=43;
		43:	DisToGoCase:=44;
		44:	// ready to receive next quedistance
			Out.ReadyForMove_PO :=1;
			//Send MCode confirmation to true
			DisToGoCase:=0;
	END_CASE

END_IF
END_METHOD

METHOD PUBLIC MoveDone : BOOL
VAR_INPUT
END_VAR
//ppr setting of hlfb is required
(*movecomplete is set either when pulsecount lines up exactly or if pulseque is empty and pulsecount is within tolerance*)
	IF Out.DistancePos_PO = Out.ExpDistancePos_PO  THEN	// (check this - add a tolerance here)
		MoveComplete :=1; 
		MoveDone := TRUE;
		busy :=0;			//set busy to zero (these are possibly interchangable until further code added) check this
		ELSE
			MoveDone :=FALSE;
		//is movedone() not completed check this
		//Add in MOVEDONE:=True; check this
	END_IF
	//movecomplete set for absolute move ppr tolerance
END_METHOD

METHOD PUBLIC Reset : BOOL
VAR_INPUT
END_VAR
//delays the turning off of reset so that it sends a full reset instead of an altspeed request
CASE ResetCase OF
	0: 
		(*Original section below for manual reset *)
		IF reset_VI =1 OR JogReset=1 THEN //reset button or auto jog reset [see jog method]
		EnableOut_FO :=0;	//Turn off to reset (power on will finish reset)
		Cancelled :=0;	//reset the cancelled move bit
		busy :=0;	// check this (is reseting busy needed?)
		DisToGoCase:=0;
		bMove_PI:=0;
		ResetCase :=10;
		OUt.MechTypeMsg_VO 		:= '';		
		Out.ConfigMSG_VO		:= '';		
		Out.ErrorMsg_VO			:= '';	
		Out.Error2Msg_VO		:= '';	
		Out.Error3Msg_VO		:='';		
		Out.Error4Msg_VO 		:='';
		Out.HomeMsg_VO 			:='';				
		OUt.LimitsMsg_VO		:='';	
		Out.ABSMoveMsg_VO		:='';
		OUt.SuperJogMsg_VO		:='';
		Out.DisToGoMsg_VO		:='';
		Out.CanceledMsg_VO		:='';
		Out.ModeMsg_VO			:='';
		LastDistanceposReq := Out.DistancePos_PO; //get rid of req diff from curr pos
		END_IF
		(*original section above for manual reset *)
	10: ResetCase:=20;
	20: ResetCase:=30;
	30: ResetCase:=40;
	40: ResetCase:=50;
	50: ResetCase:=60;
	60: ResetCase:=70;
	70: ResetCase:=80;
	80: ResetCase:=90;
	90: 
		ResetCase:=0;
		Reset_Vi:=0;
		JogReset:=0;
	
END_CASE
//reset by turning power off and then on
END_METHOD

METHOD PUBLIC SendPulse : BOOL
VAR_INPUT
END_VAR
//got rid of 'and busy =0'
IF Stop_PI = 0  AND EnableOut_FO =1 AND CW = bInputBCom_FI THEN	//check for the motor being on before incrementing the distancepos from disreq	
	IF InputAOut_FO =1  THEN 
		InputAOut_FO := 0;
	ELSE 
		IF AltSpeedReq THEN
			IF AltspeedCase =60 THEN
				InputAOut_FO :=1;		//else turn true and subtract increment counter
				AltspeedCase :=0;	//reset altspeed
				IF CW =1 THEN Out.ExpDistancePos_PO := Out.ExpDistancePos_PO +1; ELSE Out.ExpDistancePos_PO := Out.ExpDistancePos_PO - 1; END_IF
				//commenting out while testing absencoder
			END_IF
		ELSE
			InputAOut_FO :=1;		//else turn true and subtract increment counter
			IF CW =1 THEN Out.ExpDistancePos_PO := Out.ExpDistancePos_PO +1; ELSE Out.ExpDistancePos_PO := Out.ExpDistancePos_PO - 1; END_IF
			//commenting out while testing absencoder
		END_IF
		MoveComplete :=0;		//set movedone to zero and await move complete
		busy		 :=1;		//set status to busy until move complete
	END_IF	
ELSE
	//InputAOut_FO := 0;		//no trigger if stopped or direction feedback failed or if motor enable is off
	//Message Saying Move is in progress
		
END_IF
END_METHOD

METHOD StopMove : BOOL
VAR_INPUT
END_VAR
(*
	JOSEPHBARTONCHANGE3-23-2023
	This method is to stop motor movement without canceling the entire process.
*)

CASE stopCase OF
	0:
		IF bStopMove THEN
			EnableOut_FO 			:= 0;						//only way to clear out overstacked increment calls is to turn enable off and then on
			Out.ExpDistancePos_PO 	:= Out.DistancePos_PO; 		//change distancePOs_PO to float if needed
			DistancePosReq_PI  		:= Out.DistancePos_PO;		// get rid of any requestd move during cancel (must recall it after cancel)
			DisToGoCase 			:= 0;						// Remove the excess distances
			PulsesToSend 			:= 0;						// Romeve pulses from the pulse buffer
			bMove_PI 				:= 0;						// no move
			AltSpeedReq 			:= FALSE;					// no altspeed
			Out.Error4Msg_VO 		:= 'Motor Move Stopped';	// debugging line to show movement stopped using this function.
			InputAOut_FO := 0;
			MoveComplete := TRUE;
			
			stopCase := stopCase + 10;
		END_IF
		
		
	// Cycle Buffering like jake did.
	// Not sure if you have to do MoveComplete := TRUE every cycle, but Just In Case.
	10: stopCase := stopCase + 10; EnableOut_FO 	:= 0; InputAOut_FO := 0;
	20: stopCase := stopCase + 10; EnableOut_FO 	:= 0; InputAOut_FO := 0;
	30: stopCase := stopCase + 10; EnableOut_FO 	:= 0; InputAOut_FO := 0;
	40: stopCase := stopCase + 10; EnableOut_FO 	:= 0; InputAOut_FO := 0;
	50: stopCase := stopCase + 10; EnableOut_FO 	:= 0; InputAOut_FO := 0;
	60: stopCase := stopCase + 10; EnableOut_FO 	:= 0; InputAOut_FO := 0; 
	70: stopCase := stopCase + 10; EnableOut_FO 	:= 0; InputAOut_FO := 0;
	80: stopCase := stopCase + 10; EnableOut_FO 	:= 0; InputAOut_FO := 0;
	90: stopCase := stopCase + 10; EnableOut_FO 	:= 0; InputAOut_FO := 0;
	
	100: // Reset Case
		MoveComplete := TRUE;
		IF GVL_SAF.DeadmanEnable THEN EnableOut_FO := 1; END_IF		// Re-enable motor to hold motors that are not on a gearbox.
		InputAOut_FO := 0;
		
		IF NOT bStopMove THEN // Reset when ready to not stop.
			stopCase := 0;
		END_IF
		
END_CASE
END_METHOD

METHOD PUBLIC SuperJog : BOOL
VAR_INPUT
END_VAR
//using this mode will disable the two sensor safety check for manual manual mode
//homing is not required to use this and as such should be used with caution
//if not 2 sensors on and not in super mode then no movement allowed
	
	//message : at least one sensor is down please check sensors.  if movement is needed enter supermanual mode
	
//else  allow manual mode  even if not all sensors are working
	//message: you are in supermanual mode and will bypass anti collision devices.  please take caution
//add software limits check this

//add software limits check this
CASE SuperJogCase OF 
	0:	//Main Jog Sequence [Also stops movement]
		IF JogSlow_VI THEN AltspeedReq :=1; ELSE AltSpeedReq :=0;   END_IF
			
		IF SuperJogExecute_VI  THEN	//if last move is done then allow for manual increment also required to be at home //check sensor check
			(*IF IN.Limit_NC_NO_CI = 0 THEN	//NC limit switch configuration
				IF bHigh_FI AND bLow_FI THEN //set direction via hmi unless on a limit switch then default to locateposition()
					IF CW_VI = 1 	THEN	CW := 1; 	ELSE CW:=0; 	END_IF
					IF bhigh_fI = 0	THEN 	CW:=0; 		END_IF
					IF bLow_FI = 0 	THEN 	CW:=1; 		END_IF
				END_IF
				ELSE	//NO limit switch configuration
					IF bHigh_FI =0 AND bLow_FI  = 0 THEN //set direction via hmi unless on a limit switch then default to locateposition()
					IF CW_VI = 1 	THEN	CW := 1; 	ELSE CW:=0; 	END_IF
					IF bhigh_fI = 1	THEN 	CW:=0; 		END_IF
					IF bLow_FI = 1 	THEN 	CW:=1; 		END_IF
				END_IF
			END_IF*)
			IF CW_VI = 1 	THEN	CW := 1; 	ELSE CW:=0; 	END_IF
			IF AltspeedReq THEN			// slowjog if altspeed is requested and wait for case 60
				IF AltspeedCase = 60 THEN
					SendPulse();
					
				END_IF
				ELSE
					SendPulse();		//send pulse for reg speed jog
			END_IF
			ELSE
				IF	SuperJogExecute_VI  = FALSE THEN		
					CancelMove();
					SuperJogCase :=10;
				END_IF
		END_IF
	10:	//
		IF SuperJogExecute_VI =TRUE THEN SuperJogCase :=0; END_IF
		
	
END_CASE
END_METHOD

END_FUNCTION_BLOCK

// ---- Machine System/PRGs/Bogie/WX_CP_Simple.TcPOU
PROGRAM WX_CP_Simple
VAR
	WX1A_Clamp : SimpleClamp;
	WX1B_Clamp : SimpleClamp;
	
	WX2A_Clamp : SimpleClamp;
	WX2B_Clamp : SimpleClamp;
	
	WX3A_Clamp : SimpleClamp;
	WX3B_Clamp : SimpleClamp;
	
	WX4A_Clamp : SimpleClamp;
	WX4B_Clamp : SimpleClamp;
END_VAR

//WX1
WX1B_Clamp(Limit_NC_NO_CI := 0);
WX1A_Clamp(Limit_NC_NO_CI := 0);

//WX2
WX2A_Clamp(Limit_NC_NO_CI := 0);
WX2B_Clamp(Limit_NC_NO_CI := 0);

//WX3
WX3A_Clamp(Limit_NC_NO_CI := 0);
WX3B_Clamp(Limit_NC_NO_CI := 0);

//WX4
WX4A_Clamp(Limit_NC_NO_CI := 0);
WX4B_Clamp(Limit_NC_NO_CI := 0);

END_PROGRAM

// ---- Machine System/FBs/CP/SimpleClamp.TcPOU
FUNCTION_BLOCK SimpleClamp
VAR_INPUT
	ClampRequest : BOOL;
	UnClampRequest : BOOL;
	Limit_NC_NO_CI : BOOL;	// Using NC limit switches =0; Using NO Limit switches =1;
	
END_VAR
VAR_OUTPUT
	
	Clamped : BOOL;
	Unclamped : BOOL;
END_VAR
VAR
	
	//HLFB_FI 			AT %I*	: BOOL;	//high level feedback 
	
	Enable_FO 				AT %Q*  : BOOL;		//Enable ClearPath
	InputAOutCW_FO  		AT %Q* 	: BOOL; 	//input A of clearpath motor, Clockwise request move output from plc
	InputBOutCCW_FO  		AT %Q* 	: BOOL; 	//input B of clearpath motor, CounterClockwise move output from plc
	
	ClampedSensorInput_FI 	AT %I* : BOOL; 
	UnclampedSensorInput_FI AT %I* : BOOL; 
	

	
END_VAR



//Move requests if limit switches are NC

IF Limit_NC_NO_CI = 0 THEN
	IF ClampRequest AND ClampedSensorInput_FI THEN
		Enable_FO := 1;
		InputBOutCCW_FO := 1; //Clamp Direction
	ELSE
		ClampRequest := 0;
	END_IF
	
	IF UnclampRequest AND UnclampedSensorInput_FI THEN
		Enable_FO := 1;
		InputAOutCW_FO := 1; //unClamp Direction
	ELSE
		UnclampRequest :=0;
	END_IF
	
	IF NOT(UnclampRequest) AND NOT(ClampRequest) THEN
		Enable_FO := 0;
		InputAOutCW_FO := 0; //unClamp Direction
		InputBOutCCW_FO := 0; //Clamp Direction
	END_IF
	
	//FB OUTPUTS
	IF NOT(ClampedSensorInput_FI) THEN
		Clamped := 1;
	ELSE
		Clamped := 0;
	END_IF
	
	
	IF NOT(UnclampedSensorInput_FI) THEN
		Unclamped := 1;
	ELSE
		Unclamped := 0;
	END_IF
	
END_IF

END_FUNCTION_BLOCK

// ---- Machine System/PRGs/Bogie/Bogie.TcPOU
PROGRAM Bogie
VAR
	SD1 : sSD;
	SD2 : sSD;
	bTestArms : BOOL; // for testing bogie abs move
	bTest : BOOL;
	SD2_DryCycleEnable : BOOL;
	SD2_DryCycleGCODE_String : STRING;
	SD2_DryCycleOnTrig : R_TRIG;
	CNC_Start_R_Trig  : R_TRIG;
	CNC_Start_TON : TON;
	CNC_Start_TON_COMMAND : BOOL;
	
	fbWX2Handler : FB_AutoMovementHandler;
	
	bBootTest : BOOL := FALSE;
END_VAR
VAR_INPUT

END_VAR
VAR PERSISTENT
	//SD2Per: NC;
END_VAR


RequestNewMolds();

fbWX2Handler(
	WX := ADR(WX_CP.WX2)
);

IF GVL_SAF.EStopOK AND GVL_HMI.AutoMode AND bBootTest THEN
	SD1_Sequence();
	
END_IF
SD1_Control(); //Must be running all of the time
SD2_Control(); //Must be running all of the time

SD1_Status();
SD2_Status();

ACTION RequestNewMolds:
// (Dis)Enable each mold station
//Request Mold in SD1 Load position 1 if done spraying both sides and bogie is out of the spray zone
IF GVL_HMI.WX1Enable AND SD1.bSpray_A_Complete AND SD1.bSpray_B_Complete AND SD1.bInSprayPos = 0 THEN
	
	GVL_CONVEYORS.GL6.BOGIE_REQUEST_LOAD_POS_1 := 1;
	
END_IF

//Request Mold in SD1 Load position 2 if done spraying both sides and bogie is out of the spray zone
IF GVL_HMI.WX2Enable AND SD1.bSpray_A_Complete AND SD1.bSpray_B_Complete AND SD1.bInSprayPos = 0 THEN
	
	GVL_CONVEYORS.GL6.BOGIE_REQUEST_LOAD_POS_2 := 1;
	
END_IF

//Request Mold in SD2 Load position 1 if done spraying both sides and bogie is out of the spray zone
IF GVL_HMI.WX3Enable AND SD2.bSpray_A_Complete AND SD2.bSpray_B_Complete AND SD2.bInSprayPos = 0 THEN
	
	GVL_CONVEYORS.GL8.BOGIE_REQUEST_LOAD_POS_1 := 1;
	
END_IF

//Request Mold in SD2 Load position 2 if done spraying both sides and bogie is out of the spray zone
IF GVL_HMI.WX4Enable AND SD2.bSpray_A_Complete AND SD2.bSpray_B_Complete AND SD2.bInSprayPos = 0 THEN
	
	GVL_CONVEYORS.GL8.BOGIE_REQUEST_LOAD_POS_2 := 1;
	
END_IF
END_ACTION

METHOD SD1_ArmsToLoadOrientation : BOOL;
END_METHOD

ACTION SD1_ArmsToTravelOrientation:
//Rotate the Bogie arms to 90 Degrees for Travel

//WX1 Arms to Travel Pos

//WX2 Arms to Travel Pos
END_ACTION

ACTION SD1_Control:
//SD1 Servo Control 
	SD1.AxisRef();

	CASE SD1.state OF

		INIT_MOVESTATE :	(* initialisation *)
			(* initialize all function blocks *)
			SD1.AxisMoveAbsolute.Execute 	:= FALSE;
			SD1.AxisReset.Execute 			:= FALSE;
			SD1.PosistionRequestAuto 		:= NULL;
				SD1.PosistionRequestManual  := NULL;
			SD1.state := ENABLE_MOVESTATE;
			SD1.AxisStop.Execute := FALSE;

		ENABLE_MOVESTATE :
			IF GVL_SAF.EStopOK THEN
				SD1.AxisPower.Enable := TRUE;
				SD1.AxisPower.Enable_Positive := TRUE;
				SD1.AxisPower.Enable_Negative := TRUE;
				IF SD1.AxisPowerOutputs.Done  THEN
					SD1.state := WAITING_FOR_COMMAND_MOVESTATE;
				ELSIF SD1.AxisPowerOutputs.Error THEN
					SD1.state := ERROR_MOVESTATE;
				END_IF
			END_IF

		WAITING_FOR_COMMAND_MOVESTATE :		(* Wait for Position request *)
			IF GVL_HMI.AutoMode AND SD1.PosistionRequestAuto <> 0 THEN //F_CheckRollerDoor(SD1.AxisReadActualPos.Position,SD1.PosistionRequestAuto,GVL_Doors.FQ3) THEN
				SD1.fTargetPosition := LINT_TO_LREAL(SD1.PosistionRequestAuto);
				SD1.state := NEWTARGETPOSITION_MOVESTATE;
			END_IF
			IF GVL_HMI.ManualMode AND SD1.PosistionRequestManual <> 0 AND GVL_SAF.DeadmanEnable THEN //AND F_CheckRollerDoor(SD1.AxisReadActualPos.Position,SD1.PosistionRequestManual,GVL_Doors.FQ3)THEN
				SD1.fTargetPosition := LINT_TO_LREAL(SD1.PosistionRequestManual);
				SD1.state := NEWTARGETPOSITION_MOVESTATE;
			ELSIF GVL_HMI.ManualMode AND SD1.PosistionRequestManual = 0 AND GVL_SAF.DeadmanEnable THEN //Jogging in manual mode only
				SD1.AxisJog( 
    			Axis			:= SD1.AxisRef,
				JogForward		:= SD1.AxisJog.JogForward,
				JogBackwards	:= SD1.AxisJog.JogBackwards,		
				Mode			:= MC_JOGMODE_CONTINOUS,
				Velocity		:= SD1.fTargetVelocity, 
    			Done			=> SD1.AxisJogOutputs.Done,
    			Busy			=> SD1.AxisJogOutputs.Busy,
    			Active			=> SD1.AxisJogOutputs.Active,
    			CommandAborted	=> SD1.AxisJogOutputs.CommandAborted,
    			Error			=> SD1.AxisJogOutputs.Error,
    			ErrorID			=> SD1.AxisJogOutputs.ErrorID
				);
				IF SD1.AxisStopOutputs.Done THEN
					SD1.state := RESET_MOVESTATE;
				END_IF
			END_IF
			
		NEWTARGETPOSITION_MOVESTATE :		(* move to target position *)
			SD1.AxisMoveAbsolute.Position := SD1.fTargetPosition;		
			SD1.AxisMoveAbsolute.Velocity := SD1.fTargetVelocity;	
			SD1.AxisMoveAbsolute.BufferMode := MC_Buffered;
			SD1.AxisMoveAbsolute.Execute := TRUE;
			IF SD1.AxisMoveAbsoluteOutputs.Done THEN
				SD1.AxisMoveAbsolute.Execute 		:= FALSE;
				//GVL_Doors.FQ2.AutoCloseRequest 		:= 1;
				SD1.PosistionRequestAuto 			:= NULL;
				SD1.PosistionRequestManual  		:= NULL;
				GVL_HMI.SD1_ManualPositionRequest 	:= 0;
				SD1.state := WAITING_FOR_COMMAND_MOVESTATE;
			ELSIF SD1.AxisMoveAbsoluteOutputs.CommandAborted OR SD1.AxisMoveAbsoluteOutputs.Error THEN
				SD1.state := ERROR_MOVESTATE;
			END_IF

		ERROR_MOVESTATE :
			IF SD1.AxisRef.Status.Error THEN
				SD1.state := RESET_MOVESTATE;	(* axis error requires reset *)
			ELSE
				SD1.state := INIT_MOVESTATE;		(* function block errors don't need a reset *)
			END_IF

		RESET_MOVESTATE :
			SD1.AxisReset.Execute := TRUE;
			IF SD1.AxisResetOutputs.Done THEN
				SD1.state := INIT_MOVESTATE;
			ELSIF SD1.AxisResetOutputs.Error THEN
				SD1.state := INIT_MOVESTATE; (* can't do anything here *)
			END_IF
	END_CASE
	
	//Disable drive 
	IF GVL_SAF.EStopOK = 0 OR GVL_HMI.NoMode OR (NOT(GVL_SAF.DeadmanEnable) AND GVL_HMI.ManualMode) THEN
		SD1.AxisPower.Enable := FALSE;
		SD1.state := ERROR_MOVESTATE;
		SD1.PosistionRequestAuto := 0;
		SD1.PosistionRequestManual := 0;
		GVL_HMI.SD1_ManualPositionRequest := 0;
	END_IF
	
	//SD1 Function Block Calls
	SD1.AxisReset(
		Axis 	:= SD1.AxisRef,
		Busy 	=> SD1.AxisResetOutputs.Busy,
		Done 	=> SD1.AxisResetOutputs.Done,
		Error 	=> SD1.AxisResetOutputs.Error,
		ErrorID => SD1.AxisResetOutputs.ErrorID
		);
		
//	SD1.AxisReadActualPos(
//		Axis	:= SD1.AxisRef,
//    	Enable	:= TRUE,
//		//Position=> SD1.AxisReadActualPos.Position,
//		Busy 	=> SD1.AxisReadActualPosOutputs.Busy,
//		Error 	=> SD1.AxisReadActualPosOutputs.Error,
//		ErrorID => SD1.AxisReadActualPosOutputs.ErrorID
//		);

	SD1.AxisPower(
    	Axis		:= SD1.AxisRef,
//		Override	:= SD1.fOverride,
   		Status		=> SD1.AxisPowerOutputs.Done,
    	Busy 		=> SD1.AxisPowerOutputs.Busy,
		Error 		=> SD1.AxisPowerOutputs.Error,
		ErrorID 	=> SD1.AxisPowerOutputs.ErrorID
		);

	SD1.AxisMoveAbsolute(
    	Axis			:= SD1.AxisRef,
    	Done			=> SD1.AxisMoveAbsoluteOutputs.Done,
    	Busy			=> SD1.AxisMoveAbsoluteOutputs.Busy,
    	Active			=> SD1.AxisMoveAbsoluteOutputs.Active,
    	CommandAborted	=> SD1.AxisMoveAbsoluteOutputs.CommandAborted,
    	Error			=> SD1.AxisMoveAbsoluteOutputs.Error,
    	ErrorID			=> SD1.AxisMoveAbsoluteOutputs.ErrorID
		);
	
	SD1.AxisStop(
    	Axis			:= SD1.AxisRef,
		Execute			:= SD1.AxisStop.Execute,
    	Done			=> SD1.AxisStopOutputs.Done,
    	Busy			=> SD1.AxisStopOutputs.Busy,
    	Active			=> SD1.AxisStopOutputs.Active,
    	CommandAborted	=> SD1.AxisStopOutputs.CommandAborted,
    	Error			=> SD1.AxisStopOutputs.Error,
    	ErrorID			=> SD1.AxisStopOutputs.ErrorID
		);
// HMI has problems with handling Enumerations it seems, so HMI Manual buttons are handled here

IF GVL_HMI.SD1_ManualPositionRequest = 1 THEN
	
	SD1.PosistionRequestManual := SprayPos;
	
ELSIF GVL_HMI.SD1_ManualPositionRequest = 2 THEN
 
	SD1.PosistionRequestManual := RollPos;
	
ELSIF GVL_HMI.SD1_ManualPositionRequest = 3 THEN
 
	SD1.PosistionRequestManual := CurePos;
END_IF
END_ACTION

ACTION SD1_Pickup:
IF GVL_HMI.WX1Enable AND SD1.bInSprayPos AND GVL_CONVEYORS.GL6.PP_LOAD_POS_1_IS_ON AND F_PartisPresent(WX1) THEN
	
	//Call pickup of WX1
	
END_IF

IF GVL_HMI.WX2Enable AND SD1.bInSprayPos AND GVL_CONVEYORS.GL6.PP_LOAD_POS_2_IS_ON AND F_PartisPresent(WX2) THEN
	 
	//Call pickup of WX2
	
END_IF
END_ACTION

ACTION SD1_Sequence:
//SD1
IF fbWX2Handler.bError THEN
	SD1.iStep := 900;
END_IF

CASE SD1.iStep OF
	

	0: //Default
		//Do nothing mode. (This means you can't have things that rely on being called EVERY cycle)
		
	10: //Move arms into load position
		fbWX2Handler.nMoveState := Load_Position;
		IF fbWX2Handler.bMoveComplete THEN		
			SD1.iStep := 20;
		END_IF
		
	20: //Drive SD to 'Pickup Position'
		IF SD1.bInPickupPos THEN
			SD1.iStep := 30;
		ELSE
			SD1.PosistionRequestAuto := PickupPos;
		END_IF
	
	30: //Clamp tool
		IF GVL_CONVEYORS.GL6.PP_Load_Pos_1_Is_On AND GVL_HMI.WX1Enable THEN
			//wx1 clamp
		END_IF
		IF GVL_CONVEYORS.GL6.PP_Load_Pos_2_Is_On AND GVL_HMI.WX2Enable THEN
			fbWX2Handler.nMoveState := CLAMP;
		END_IF
		
		IF F_PartIsPresentAndClamped(GVL_IO.WX1) AND F_PartIsPresentAndClamped(GVL_IO.WX2)  THEN 
			SD1.iStep := 40;
		END_IF
		
	40: //Move arms to lifted position
		fbWX2Handler.nMoveState := LIFTED_POSITION;
		IF fbWX2Handler.bMoveComplete THEN
			SD1.iStep := 50;
		END_IF
		
	50: //Jog SD axis to spray position
		IF SD1.bInSprayPos THEN
			SD1.iStep := 70;
		ELSE
			SD1.PosistionRequestAuto := SprayPos;
		END_IF
(*Side A ----------------------------------------------------------------*)		
	60: //Call Side A Spray
		IF PRG_CNCChannelHandler.CNCChannel[0].currentmode = 3 THEN
			PLCMachineMode[0].MDIString := WSTRING_TO_STRING("L C://CNC/TestSpray");
			PLCMachineMode[0].Start := TRUE;
			SD1.bSpray_A_Complete := 0;
		END_IF
		IF SD1.bSpray_A_Complete THEN
			SD1.iStep := 70;
		END_IF
			
	70:	//Move to Roll	
		SD1.PosistionRequestAuto := RollPos;
		IF SD1.bInRollPos THEN 	
			SD1.iStep := 80;
		END_IF
		
	80: //Side A Roll
		IF SD1.bRoll_A_Complete  THEN
			SD1.iStep := 90;
		END_IF
			
	90: //Side A Place Ribs if required It's a database check. From the data in the data structure in the PLC.
		IF SD1.bPlace_A_Complete THEN 
			SD1.iStep := 100;
		END_IF

	100: //Move to Cure
		SD1.PosistionRequestAuto := CurePos;
		IF SD1.bInCurePos THEN
		 	SD1.iStep := 110;
		END_IF	

	110: //Side A Cure
		//Start Heater here 
		IF SD1.bCure_A_Complete THEN
		 	SD1.iStep := 120;
		END_IF
		
(*Side B -----------------------------------------------------------*)
		
	120: //Move to Spray WX Side B & SD
		SD1.PosistionRequestAuto := SprayPos;
		IF SD1.bInSprayPos THEN
			SD1.iStep := 130;
		END_IF
		
	130: //Side B Spray
		IF PRG_CNCChannelHandler.CNCChannel[0].currentmode = 3 THEN
			PLCMachineMode[0].MDIString := WSTRING_TO_STRING("L C://CNC/TestSpray");
			PLCMachineMode[0].Start := TRUE;
			SD1.bSpray_B_Complete := 0;
		END_IF
		IF SD1.bSpray_B_Complete THEN
			SD1.iStep := 135;
		END_IF
			
	135: //Move to Roll
		SD1.PosistionRequestAuto := RollPos;
		IF SD1.bInRollPos THEN 
			SD1.iStep := 140;
		END_IF
		
	140: //Side B Roll
		IF SD1.bRoll_B_Complete  THEN
			SD1.iStep := 150;
		END_IF
			
	150: //Side B Place
		IF SD1.bPlace_B_Complete THEN 
			SD1.iStep := 160;
		END_IF
		
	160: //Move to Cure
		SD1.PosistionRequestAuto := CurePos;
		IF SD1.bInCurePos THEN 
			SD1.iStep := 170;
		END_IF
		
	170: //Side B Cure
		IF SD1.bCure_B_Complete  THEN
			SD1.iStep := 180;
		END_IF
(*
		When the cure is complete, and the putdown zone is not clear, then we need to have a space to keep the arms that is not under the heaters.
			we could over-cure the mold.
			
			For now keep in roll position until the putdown position is clear. (after side B RIB placement)
*)

	(* Move To Putdown & Lifted Position -------------------------------------------------------------------------------------*)
	
	180:	//move to PutDownPos
		IF SD1.bPutDownZoneClear AND fbWX2Handler.nMoveState = STANDBY THEN
			SD1.PosistionRequestAuto := PutDownPos;
			fbWX2Handler.nMoveState := LIFTED_POSITION;
			SD1.iStep := 190;
		END_IF
	190: // Waiting for motor movement completion
		IF SD1.bInPutDownPos AND (NOT fbWX2Handler.nMoveState = LIFTED_POSITION AND fbWX2Handler.bMoveComplete) THEN
			SD1.iStep := 170;
		END_IF
	
	
	(* Arms To Unload Position & Unclamp -------------------------------------------------------------------------------------------*)
		
	170: //Set Down Molds
		IF NOT fbWX2Handler.nMoveState = UNLOAD_POSITION AND NOT fbWX2Handler.bBusy THEN
			fbWX2Handler.nMoveState := UNLOAD_POSITION;
			SD1.iStep := 171;
		END_IF
	171: // Wait for motor movement completion, and then unclamp motor.
		IF NOT fbWX2Handler.nMoveState = UNLOAD_POSITION AND fbWX2Handler.bMoveComplete THEN
			fbWX2Handler.nMoveState := UNCLAMP;
			SD1.iStep := 172;
		END_IF
	172: // Wait for unclamp to finish
		IF NOT fbWX2Handler.nMoveState = UNCLAMP AND fbWX2Handler.bMoveComplete AND NOT fbWX2Handler.bClamped THEN
			SD1.iStep := 180;
		END_IF
		
	(* Backup Traverse, and Arms To Travel Orientation ------------------------------------------------------------------------*)
		
	180: //Move to PostPutDownPos
		SD1.PosistionRequestAuto := PostPutDownPos;
		IF SD1.bInPostPutDownPos AND NOT fbWX2Handler.bClamped THEN
			SD1.iStep := 185; 
		END_IF
		
	185: //Rotate Clamp Arms to Travel Position 90 degrees
		IF NOT fbWX2Handler.bClamped AND SD1.bInPostPutDownPos THEN
			fbWX2Handler.nMoveState := TRAVERSE_POSITION;
			SD1.iStep := 186;
		END_IF
	186: // Waiting for motor movement completion
		IF NOT fbWX2Handler.nMoveState = TRAVERSE_POSITION AND fbWX2Handler.bMoveComplete THEN
			SD1.iStep := 190;
		END_IF
		
	(* Move to start of spray line to pick up next Tool ------------------------------------------------------------------------------------------------*)
	
	190: //Move to Pre Pick up Pos
		IF NOT fbWX2Handler.bBusy THEN 
			SD1.PosistionRequestAuto := PrePickupPos;
		END_IF
		
		IF SD1.bInPrePickupPos THEN 
			SD1.iStep := 3;
		END_IF
		
	(* Errors ------------------------------------------------------------------------------------------------------------------------------------------*)
		
	900: //errors
		IF fbWX2Handler.bError THEN
			SD1.sWXErrorMessage := fbWX2Handler.sErrorMessage;
			SD1.bWXError 		:= TRUE;
		END_IF
		
		IF SD1.bSDError THEN
			SD1.bSDError := TRUE; 
		END_IF
		
END_CASE
END_ACTION

ACTION SD1_SetDown:
IF SD1.bInPutDownPos AND SD1.bPutDownZoneClear AND (GVL_IO.WX1.A.bPP1_Input OR GVL_IO.WX1.A.bPP2_Input OR GVL_IO.WX1.B.bPP1_Input OR GVL_IO.WX1.B.bPP2_Input) THEN
	
	//Call Putdown of WX1
	
END_IF

IF SD1.bInPutDownPos AND SD1.bPutDownZoneClear AND (GVL_IO.WX2.A.bPP1_Input OR GVL_IO.WX2.A.bPP2_Input OR GVL_IO.WX2.B.bPP1_Input OR GVL_IO.WX2.B.bPP2_Input) THEN
	
	//Call Putdown of WX2
	
END_IF
END_ACTION

ACTION SD1_Status:
//Position Window Variables

	SD1.fSprayPosWindowMin		:= SprayPos - SD1.fPosTolerance;
	SD1.fSprayPosWindowMax		:= SprayPos + SD1.fPosTolerance;
	
	SD1.fPrePickupPosWindowMin	:= PrePickupPos - SD1.fPosTolerance;
	SD1.fPrePickupPosWindowMax	:= PrePickupPos + SD1.fPosTolerance;
	
	SD1.fRollPosWindowMin		:= RollPos - SD1.fPosTolerance;
	SD1.fRollPosWindowMax		:= RollPos + SD1.fPosTolerance;

	SD1.fCurePosWindowMin		:= CurePos - SD1.fPosTolerance;
	SD1.fCurePosWindowMax		:= CurePos + SD1.fPosTolerance;

	SD1.fPutDownPosWindowMin 	:= PutDownPos - SD1.fPosTolerance;
	SD1.fPutDownPosWindowMax 	:= PutDownPos + SD1.fPosTolerance;
	
//Position status - check if either in Spray, Roll, or Cure Zone 

	//PREPICKUP POS
	IF SD1.AxisReadActualPos.Position > SD1.fPrePickupPosWindowMin AND
	   SD1.AxisReadActualPos.Position < SD1.fPrePickupPosWindowMax THEN
		SD1.bInPrePickupPos := 1;
	ELSE
		SD1.bInPrePickupPos := 0;
	END_IF
	//SPRAY/PICKUP POS
	IF SD1.AxisReadActualPos.Position > SD1.fSprayPosWindowMin AND
	   SD1.AxisReadActualPos.Position < SD1.fSprayPosWindowMax THEN
		SD1.bInSprayPos := 1;
	ELSE
		SD1.bInSprayPos := 0;
	END_IF
	//ROLL POS
	IF SD1.AxisReadActualPos.Position	> SD1.fRollPosWindowMin AND
	   SD1.AxisReadActualPos.Position < SD1.fRollPosWindowMax THEN
		SD1.bInRollPos := 1;
	ELSE
		SD1.bInRollPos := 0;
	END_IF
	//CURE POS
	IF SD1.AxisReadActualPos.Position > SD1.fCurePosWindowMin AND
	   SD1.AxisReadActualPos.Position < SD1.fCurePosWindowMax THEN
		SD1.bInCurePos := 1;
	ELSE
		SD1.bInCurePos := 0;
	END_IF
	//PUTDOWN POS
	IF SD1.AxisReadActualPos.Position > SD1.fPutDownPosWindowMin AND
	   SD1.AxisReadActualPos.Position < SD1.fPutDownPosWindowMax THEN
		SD1.bInPutDownPos := 1;
	ELSE
		SD1.bInPutDownPos := 0;
	END_IF

//Conveyor Inputs
GVL_IO.WX1.ConveyorLoadPos := GVL_CONVEYORS.GL6.PP_LOAD_POS_1_IS_ON; 
GVL_IO.WX2.ConveyorLoadPos := GVL_CONVEYORS.GL6.PP_LOAD_POS_2_IS_ON; 

//HMI Inputs to Bogie Structure
GVL_IO.WX1.bEnabled := GVL_HMI.WX1Enable;
GVL_IO.WX2.bEnabled := GVL_HMI.WX2Enable;

//Status from CNC
SD1.bSpray_A_Complete 	:= CNCSystem.Channel[0].M[570].bState_rw; 
SD1.bRoll_A_Complete 	:= CNCSystem.Channel[0].M[571].bState_rw;
SD1.bPlace_A_Complete 	:= CNCSystem.Channel[0].M[572].bState_rw;

SD1.bSpray_B_Complete 	:= CNCSystem.Channel[0].M[573].bState_rw; 
SD1.bRoll_B_Complete 	:= CNCSystem.Channel[0].M[574].bState_rw;
SD1.bPlace_B_Complete 	:= CNCSystem.Channel[0].M[575].bState_rw;
END_ACTION

ACTION SD2_ArmsToLoadOrientation:
//Rotate the Bogie arms to 0 Degrees for Picking up part

//WX3 Arms to 0 degrees

//WX4 Arms to 0 degrees
END_ACTION

ACTION SD2_ArmsToTravelOrientation:
//Rotate the Bogie arms to 90 Degrees for Travel

//WX3 Arms to Travel Pos

//WX4 Arms to Travel Pos
END_ACTION

ACTION SD2_Control:
//SD2 Servo Control 
	SD2.AxisRef();

	CASE SD2.state OF

		INIT_MOVESTATE :	(* initialisation *)
			(* initialize all function blocks *)
			SD2.AxisMoveAbsolute.Execute 	:= FALSE;
			SD2.AxisReset.Execute 			:= FALSE;
			SD2.PosistionRequestAuto 		:= NULL;
				SD2.PosistionRequestManual  := NULL;
			SD2.state := ENABLE_MOVESTATE;
			SD2.AxisStop.Execute := FALSE;

		ENABLE_MOVESTATE :
			IF GVL_SAF.EStopOK THEN
				SD2.AxisPower.Enable := TRUE;
				SD2.AxisPower.Enable_Positive := TRUE;
				SD2.AxisPower.Enable_Negative := TRUE;
				IF SD2.AxisPowerOutputs.Done  THEN
					SD2.state := WAITING_FOR_COMMAND_MOVESTATE;
				ELSIF SD2.AxisPowerOutputs.Error THEN
					SD2.state := ERROR_MOVESTATE;
				END_IF
			END_IF

		WAITING_FOR_COMMAND_MOVESTATE :		(* Wait for Position request *)
			IF GVL_HMI.AutoMode AND SD2.PosistionRequestAuto <> 0 THEN //F_CheckRollerDoor(SD2.AxisReadActualPos.Position,SD2.PosistionRequestAuto,GVL_Doors.FQ3) THEN
				SD2.fTargetPosition := LINT_TO_LREAL(SD2.PosistionRequestAuto);
				SD2.state := NEWTARGETPOSITION_MOVESTATE;
			END_IF
			IF GVL_HMI.ManualMode AND SD2.PosistionRequestManual <> 0 AND GVL_SAF.DeadmanEnable THEN //AND F_CheckRollerDoor(SD2.AxisReadActualPos.Position,SD2.PosistionRequestManual,GVL_Doors.FQ3)THEN
				SD2.fTargetPosition := LINT_TO_LREAL(SD2.PosistionRequestManual);
				SD2.state := NEWTARGETPOSITION_MOVESTATE;
			ELSIF GVL_HMI.ManualMode AND SD2.PosistionRequestManual = 0 AND GVL_SAF.DeadmanEnable THEN //Jogging in manual mode only
				SD2.AxisJog( 
    			Axis			:= SD2.AxisRef,
				JogForward		:= SD2.AxisJog.JogForward,
				JogBackwards	:= SD2.AxisJog.JogBackwards,		
				Mode			:= MC_JOGMODE_CONTINOUS,
				Velocity		:= SD2.fTargetVelocity, 
    			Done			=> SD2.AxisJogOutputs.Done,
    			Busy			=> SD2.AxisJogOutputs.Busy,
    			Active			=> SD2.AxisJogOutputs.Active,
    			CommandAborted	=> SD2.AxisJogOutputs.CommandAborted,
    			Error			=> SD2.AxisJogOutputs.Error,
    			ErrorID			=> SD2.AxisJogOutputs.ErrorID
				);
				IF SD2.AxisStopOutputs.Done THEN
					SD2.state := RESET_MOVESTATE;
				END_IF
			END_IF
			
		NEWTARGETPOSITION_MOVESTATE :		(* move to target position *)
			SD2.AxisMoveAbsolute.Position := SD2.fTargetPosition;		
			SD2.AxisMoveAbsolute.Velocity := SD2.fTargetVelocity;	
			SD2.AxisMoveAbsolute.BufferMode := MC_Buffered;
			SD2.AxisMoveAbsolute.Execute := TRUE;
			IF SD2.AxisMoveAbsoluteOutputs.Done THEN
				SD2.AxisMoveAbsolute.Execute 		:= FALSE;
				GVL_Doors.FQ2.AutoCloseRequest 		:= 1;
				SD2.PosistionRequestAuto 			:= NULL;
				SD2.PosistionRequestManual  		:= NULL;
				GVL_HMI.SD2_ManualPositionRequest 	:= 0;
				SD2.state := WAITING_FOR_COMMAND_MOVESTATE;
			ELSIF SD2.AxisMoveAbsoluteOutputs.CommandAborted OR SD2.AxisMoveAbsoluteOutputs.Error THEN
				SD2.state := ERROR_MOVESTATE;
			END_IF

		ERROR_MOVESTATE :
			IF SD2.AxisRef.Status.Error THEN
				SD2.state := RESET_MOVESTATE;	(* axis error requires reset *)
			ELSE
				SD2.state := INIT_MOVESTATE;		(* function block errors don't need a reset *)
			END_IF

		RESET_MOVESTATE :
			SD2.AxisReset.Execute := TRUE;
			IF SD2.AxisResetOutputs.Done THEN
				SD2.state := INIT_MOVESTATE;
			ELSIF SD2.AxisResetOutputs.Error THEN
				SD2.state := INIT_MOVESTATE; (* can't do anything here *)
			END_IF
	END_CASE
	
	//Disable drive 
	IF GVL_SAF.EStopOK = 0 OR GVL_HMI.NoMode OR (NOT(GVL_SAF.DeadmanEnable) AND GVL_HMI.ManualMode) THEN
		SD2.AxisPower.Enable := FALSE;
		SD2.state := ERROR_MOVESTATE;
		SD2.PosistionRequestAuto := 0;
		SD2.PosistionRequestManual := 0;
		GVL_HMI.SD2_ManualPositionRequest := 0;
	END_IF
	
	//SD2 Function Block Calls
	SD2.AxisReset(
		Axis 	:= SD2.AxisRef,
		Busy 	=> SD2.AxisResetOutputs.Busy,
		Done 	=> SD2.AxisResetOutputs.Done,
		Error 	=> SD2.AxisResetOutputs.Error,
		ErrorID => SD2.AxisResetOutputs.ErrorID
		);
		
//	SD2.AxisReadActualPos(
//		Axis	:= SD2.AxisRef,
//    	Enable	:= TRUE,
//		//Position=> SD2.AxisReadActualPos.Position,
//		Busy 	=> SD2.AxisReadActualPosOutputs.Busy,
//		Error 	=> SD2.AxisReadActualPosOutputs.Error,
//		ErrorID => SD2.AxisReadActualPosOutputs.ErrorID
//		);

	SD2.AxisPower(
    	Axis		:= SD2.AxisRef,
//		Override	:= SD2.fOverride,
   		Status		=> SD2.AxisPowerOutputs.Done,
    	Busy 		=> SD2.AxisPowerOutputs.Busy,
		Error 		=> SD2.AxisPowerOutputs.Error,
		ErrorID 	=> SD2.AxisPowerOutputs.ErrorID
		);

	SD2.AxisMoveAbsolute(
    	Axis			:= SD2.AxisRef,
    	Done			=> SD2.AxisMoveAbsoluteOutputs.Done,
    	Busy			=> SD2.AxisMoveAbsoluteOutputs.Busy,
    	Active			=> SD2.AxisMoveAbsoluteOutputs.Active,
    	CommandAborted	=> SD2.AxisMoveAbsoluteOutputs.CommandAborted,
    	Error			=> SD2.AxisMoveAbsoluteOutputs.Error,
    	ErrorID			=> SD2.AxisMoveAbsoluteOutputs.ErrorID
		);
	
	SD2.AxisStop(
    	Axis			:= SD2.AxisRef,
		Execute			:= SD2.AxisStop.Execute,
    	Done			=> SD2.AxisStopOutputs.Done,
    	Busy			=> SD2.AxisStopOutputs.Busy,
    	Active			=> SD2.AxisStopOutputs.Active,
    	CommandAborted	=> SD2.AxisStopOutputs.CommandAborted,
    	Error			=> SD2.AxisStopOutputs.Error,
    	ErrorID			=> SD2.AxisStopOutputs.ErrorID
		);
// HMI has problems with handling Enumerations it seems, so HMI Manual buttons are handled here

IF GVL_HMI.SD2_ManualPositionRequest = 1 THEN
	
	SD2.PosistionRequestManual := SprayPos;
	
ELSIF GVL_HMI.SD2_ManualPositionRequest = 2 THEN
 
	SD2.PosistionRequestManual := RollPos;
	
ELSIF GVL_HMI.SD2_ManualPositionRequest = 3 THEN
 
	SD2.PosistionRequestManual := CurePos;
END_IF
END_ACTION

ACTION SD2_DryCycle:
//SD2

CNC_Start_TON(IN:=CNC_Start_TON_COMMAND,PT:=T#2500MS);

SD2_DryCycleOnTrig(CLK :=SD2_DryCycleEnable);
	IF SD2_DryCycleOnTrig.Q THEN
		SD2.iStepDry := 1;
		
		END_IF
		

IF SD2_DryCycleEnable THEN
	

	Global_HMI.PLCMachineMode[0].MDI := 1;
	Global_HMI.PLCMachineMode[0].ManualMode.nManualTyp := 1;


	CASE SD2.iStepDry OF
//	0: 	//default
	1: SD2.PosistionRequestAuto := SprayPos;
	IF SD2.bInSprayPos 	 THEN 	SD2.iStepDry := 25;	END_IF
    5:	//Check that WX1 and WX2 are empty and do not contain a mold, then rotate arms to Load Orientation
		IF SD2.bInPrePickupPos THEN
			SD2_ArmsToLoadOrientation();
		END_IF
		SD2.iStepDry := 10;
	10: //Move to Spray/Pickup Pos
		IF SD2.bInPrePickupPos THEN
			SD2.PosistionRequestAuto := SprayPos;				
		END_IF
		IF SD2.bInSprayPos 	 THEN 	SD2.iStepDry := 15;	END_IF
	15: //Check if there there molds ready for pickup and pickup if mold present and WX is enabled
		IF SD2.bInSprayPos THEN SD2.iStepDry := 25; END_IF
//	17: 
//		CNC_Start_TON_COMMAND := 1;
//		SD2.iStepDry := 20;
		
//	20: //Side A Spray

//		IF PRG_CNCChannelHandler.CNCChannel[0].currentmode = 3 THEN
//			PLCMachineMode[0].MDIString := 'G01 X1700 F9000 
//G01 Y4000 F5000
//G01 X1400 F9000
//G01 Y2000 F5000';
			

//			IF CNC_Start_TON.ET < T#2500MS AND CNC_Start_TON.ET > T#0MS THEN
//				PLCMachineMode[0].Start := TRUE;
//			END_IF
//			IF CNC_Start_TON.Q THEN
//				CNC_Start_TON_COMMAND := 0;
//				PLCMachineMode[0].Start := FALSE;
			
//			END_IF
		
//		END_IF
		
//		IF Global_HMI.PLCMachineMode[0].Ready = 1 THEN	SD2.iStepDry := 25;	END_IF
	25:	//Move to Roll	
		SD2.PosistionRequestAuto := RollPos;
		IF SD2.bInRollPos  THEN 	SD2.iStepDry := 190;	END_IF
	190: //Move to Pre Pick up Pos
		
		SD2.PosistionRequestAuto := PrePickupPos;
		
		IF SD2.bInPrePickupPos THEN SD2.iStepDry := 5; END_IF
	END_CASE
END_IF
END_ACTION

ACTION SD2_Pickup:
IF GVL_HMI.WX3Enable AND SD1.bInSprayPos AND GVL_CONVEYORS.GL6.PP_LOAD_POS_1_IS_ON AND F_PartisPresent(WX3) THEN
	
	//Call pickup of WX3
	
END_IF

IF GVL_HMI.WX4Enable AND SD1.bInSprayPos AND GVL_CONVEYORS.GL6.PP_LOAD_POS_2_IS_ON AND F_PartisPresent(WX4) THEN
	 
	//Call pickup of WX4
	
END_IF
END_ACTION

ACTION SD2_Sequence:
//SD2
	(* seq begins when 2 molds are picked up.  Their GCode file 'strings' should be stored in RFID Tag *)
	//Call PickupSD2()
	//Add Mold Job Files to Spray Que [FIFO] 
		//WX1:Key_A, WX1:Macro_A, WX2:Key_A, WX2:Macro_A, WX1:Key_B, WX1:Macro_B, WX2:Key_B, WX2:Macro_B
	//Add Mold Job Files to Roll Que [FIFO]
		//WX1:Key_A, WX1:Macro_A, WX2:Key_A, WX2:Macro_A, SoftCureSideA, WX1:Key_B, WX1:Macro_B, WX2:Key_B, WX2:Macro_B, SOFTCureSideB
	//Add Mold Job Files to Place Que [FIFO] (*These will prob need a FIFO Priority but allow for opportunity running on SD2*)
		//WX1:Side_A, WX2:Side_A, WX1:Side_B, WX2:Side_B 
	//Await Job Complete then --- Call SetDownSD2()
	//SD2 Case
	CASE SD2.iStep OF
	0: 	//default
	5:	//Check that WX1 and WX2 are empty and do not contain a mold, then rotate arms to Load Orientation
		IF F_IsEmpty(WX1) = 0 AND F_IsEmpty(WX2) AND SD2.bInPrePickupPos THEN
			SD2_ArmsToLoadOrientation();
		END_IF
		SD2.iStep := 10;
	10: //Move to Spray/Pickup Pos
		IF SD2.bInPrePickupPos AND F_ArmsInLoadOrientation() THEN
			SD2.PosistionRequestAuto := SprayPos;				
		END_IF
		IF SD2.bInSprayPos 		 THEN 	SD2.iStep := 15;	END_IF
	15: //Check if there there molds ready for pickup and pickup if mold present and WX is enabled
		IF SD2.bInSprayPos THEN SD2_Pickup(); END_IF
	
		IF F_PartPickupSuccess(WX1) AND F_PartPickupSuccess(WX2) THEN
			SD2.iStep := 17;
			ELSE
			SD2.iStep := 0;
			//No Mold to pick up 
		END_IF
	17: //Add Files to Que
		IF F_PartIsPresent(WX1) THEN
			//Get mold id and Database data and put into WX1.CurrentJob
			//Load files for WX1 
			WX1.CurrentJob.AKeyFile := 'test.nc';
		END_IF
		IF F_PartIsPresent(WX2) THEN
			//Load files for WX2
			WX2.CurrentJob.AKeyFile := 'test2.nc';
			//Get mold id and Database data and put into WX2.CurrentJob
		END_IF
		//check if files present and loaded
		IF F_CheckMoldData(WX1.CurrentJob.MoldID,GVL_HMI.WX1Enable) AND F_CheckMoldData(WX1.CurrentJob.MoldID,GVL_HMI.WX1Enable) THEN
			SD2.iStep := 20;
			ELSE
				//Mold Data missing or incorrect
		END_IF
	20: //Side A Spray
		IF SD2.bSpray_A_Complete THEN	SD2.iStep := 25;	END_IF
	25:	//Move to Roll	
		SD2.PosistionRequestAuto := RollPos;
		IF SD2.bInRollPos 		 THEN 	SD2.iStep := 30;	END_IF
	30: //Side A Roll
		IF SD2.bRoll_A_Complete  THEN	SD2.iStep := 40;	END_IF
	40: //Side A Place
		IF SD2.bPlace_A_Complete THEN 	SD2.iStep := 45;	END_IF
	45: //Move to Cure
		SD2.PosistionRequestAuto := CurePos;
		IF SD2.bInCurePos 		 THEN 	SD2.iStep := 50;	END_IF
	50: //Side A Cure
		IF SD2.bCure_A_Complete  THEN 	SD2.iStep := 55;	END_IF
	55: //Move to Spray
		SD2.PosistionRequestAuto := SprayPos;
		IF SD2.bInSprayPos 		 THEN 	SD2.iStep := 120;	END_IF
	120: //Side B Spray
		IF SD2.bSpray_B_Complete THEN	SD2.iStep := 125;	END_IF
	125: //Move to Roll
		SD2.PosistionRequestAuto := RollPos;
		IF SD2.bInRollPos 		 THEN 	SD2.iStep := 130;	END_IF
	130: //Side B Roll
		IF SD2.bRoll_B_Complete  THEN	SD2.iStep := 140;	END_IF
	140: //Side B Place
		IF SD2.bPlace_B_Complete THEN 	SD2.iStep := 145;	END_IF
	145: //Move to Cure
		SD2.PosistionRequestAuto := CurePos;
		IF SD2.bInCurePos 		 THEN 	SD2.iStep := 150;	END_IF
	150: //Side B Cure
		IF SD2.bCure_B_Complete  THEN	SD2.iStep := 165;	END_IF
	165:	//move to PutDownPos
		IF SD2.bPutDownZoneClear THEN
			SD2.PosistionRequestAuto := PutDownPos;
		END_IF
		IF SD2.bInPutDownPos 	 THEN 	SD2.iStep := 170;	END_IF
	170: //Set Down Molds
		IF SD2.bJob_Complete	THEN
			SD2_SetDown(); 
		END_IF
	180: //Move to PostPutDownPos
		IF WX1.A.bClampLimitLow AND WX1.B.bClampLimitLow AND 
		   WX2.A.bClampLimitLow AND WX2.B.bClampLimitLow THEN
			SD2.PosistionRequestAuto := PostPutDownPos;
		END_IF
		IF SD2.bInPostPutDownPos AND F_IsEmpty(WX1) AND F_IsEmpty(WX2)  THEN SD2.iStep := 185; END_IF
	185: //Rotate Clamp Arms to Travel Position 90 degrees
		SD2_ArmsToTravelOrientation();
		IF WX1.bArmsAtTravelPos AND WX2.bArmsAtTravelPos THEN SD2.iStep := 190;	END_IF
	190: //Move to Pre Pick up Pos
		IF WX1.bArmsAtTravelPos AND WX2.bArmsAtTravelPos THEN 
			SD2.PosistionRequestAuto := PrePickupPos;
			ELSE
				SD2_ArmsToTravelOrientation();
		END_IF
		
		IF SD2.bInPrePickupPos THEN SD2.iStep := 5; END_IF
	900: //errors
	END_CASE
END_ACTION

ACTION SD2_SetDown:
IF SD2.bInPutDownPos AND SD2.bPutDownZoneClear AND (GVL_IO.WX3.A.bPP1_Input OR GVL_IO.WX3.A.bPP2_Input OR GVL_IO.WX3.B.bPP1_Input OR GVL_IO.WX3.B.bPP2_Input) THEN
	
	//Call Putdown of WX3
	
END_IF

IF SD2.bInPutDownPos AND SD2.bPutDownZoneClear AND (GVL_IO.WX4.A.bPP1_Input OR GVL_IO.WX4.A.bPP2_Input OR GVL_IO.WX4.B.bPP1_Input OR GVL_IO.WX4.B.bPP2_Input) THEN
	
	//Call Putdown of WX4
	
END_IF
END_ACTION

ACTION SD2_Status:
//Position Window Variables

	SD2.fSprayPosWindowMin		:= SprayPos - SD2.fPosTolerance;
	SD2.fSprayPosWindowMax		:= SprayPos + SD2.fPosTolerance;
	
	SD2.fPrePickupPosWindowMin	:= PrePickupPos - SD2.fPosTolerance;
	SD2.fPrePickupPosWindowMax	:= PrePickupPos + SD2.fPosTolerance;
	
	SD2.fRollPosWindowMin		:= RollPos - SD2.fPosTolerance;
	SD2.fRollPosWindowMax		:= RollPos + SD2.fPosTolerance;
	
	SD2.fCurePosWindowMin		:= CurePos - SD2.fPosTolerance;
	SD2.fCurePosWindowMax		:= CurePos + SD2.fPosTolerance;

	SD2.fPutDownPosWindowMin 	:= PutDownPos - SD2.fPosTolerance;
	SD2.fPutDownPosWindowMax 	:= PutDownPos + SD2.fPosTolerance;
	
//Position status - check if either in Spray, Roll, or Cure Zone 

	//PREPICKUP POS
	IF SD2.AxisReadActualPos.Position > SD2.fPrePickupPosWindowMin AND
	   SD2.AxisReadActualPos.Position < SD2.fPrePickupPosWindowMax THEN
		SD2.bInPrePickupPos := 1;
	ELSE
		SD2.bInPrePickupPos := 0;
	END_IF
	//SPRAY/PICKUP POS
	IF SD2.AxisReadActualPos.Position > SD2.fSprayPosWindowMin AND
	   SD2.AxisReadActualPos.Position < SD2.fSprayPosWindowMax THEN
		SD2.bInSprayPos := 1;
	ELSE
		SD2.bInSprayPos := 0;
	END_IF
	//ROLL POS
	IF SD2.AxisReadActualPos.Position	> SD2.fRollPosWindowMin AND
	   SD2.AxisReadActualPos.Position < SD2.fRollPosWindowMax THEN
		SD2.bInRollPos := 1;
	ELSE
		SD2.bInRollPos := 0;
	END_IF
	//CURE POS
	IF SD2.AxisReadActualPos.Position > SD2.fCurePosWindowMin AND
	   SD2.AxisReadActualPos.Position < SD2.fCurePosWindowMax THEN
		SD2.bInCurePos := 1;
	ELSE
		SD2.bInCurePos := 0;
	END_IF
	//PUTDOWN POS
	IF SD2.AxisReadActualPos.Position > SD2.fPutDownPosWindowMin AND
	   SD2.AxisReadActualPos.Position < SD2.fPutDownPosWindowMax THEN
		SD2.bInPutDownPos := 1;
	ELSE
		SD2.bInPutDownPos := 0;
	END_IF

//Conveyor Inputs
GVL_IO.WX3.ConveyorLoadPos := GVL_CONVEYORS.GL6.PP_LOAD_POS_1_IS_ON; //JosephBartonChange1-11-2023 I made these both the proper WX3&4 instead of 1&2
GVL_IO.WX4.ConveyorLoadPos := GVL_CONVEYORS.GL6.PP_LOAD_POS_2_IS_ON; //JosephBartonChange1-11-2023 

//HMI Inputs to Bogie Structure
GVL_IO.WX3.bEnabled := GVL_HMI.WX3Enable; //JosephBartonChange1-11-2023 I also made these the proper WX3&4 instead of 1&2
GVL_IO.WX4.bEnabled := GVL_HMI.WX4Enable; //JosephBartonChange1-11-2023
END_ACTION

END_PROGRAM

// ---- Machine System/FBs/FB_AutoMovementHandler.TcPOU
FUNCTION_BLOCK FB_AutoMovementHandler
VAR_INPUT
	// Bogie arms to use
	WX : POINTER TO BogieComboWX;
	
	// State Handler case
	nMoveState : eBogieHandlerCase := STANDBY;
END_VAR
	
VAR_OUTPUT
	//Status Variables
	bMoveComplete : BOOL 		:= FALSE;
	bBusy 		  : BOOL 		:= FALSE; // While bBusy := TRUE; assume motor movement.
	bClamped	  : BOOL 		:= FALSE;
	bHomed    	  : BOOL		:= FALSE;
	
	// Error Variables
	bError 		  : BOOL 		:= FALSE;
	sErrorMessage : STRING(255) := '';
	
	bTest : BOOL;
END_VAR

VAR
	// Bogie arm target position
	WX2TargetPos : sBogieArmPosition;
	
	//Clamp Error Detection
	nWX2ClampedAPos	: LREAL;
	nWX2ClampedBPos : LREAL;
	nClampTolerance : INT := 2;
	
	//Timeout Error Detection
	tStartTime : TIME;
	tTimeLimit : TIME := T#45S;
	
	// General Vars
	nCounter : USINT := 0;
	
	//Initialising Variables
	bInit 	 : BOOL := FALSE;
	
	//Motor Movement Variables
	bCleanUp 			: BOOL := FALSE;
	bCleanUpBusy		: BOOL := FALSE;
	bInitCleanUpTrigger : BOOL := FALSE;
	
	//Clamping Variables
	nClamp_ATracker : ARRAY[1..100] OF REAL;
	nClamp_BTracker : ARRAY[1..100] OF REAL;
		
	nClampAvgPos	: REAL;
	nClampCounter : INT := 1;	// Don't use me.
	
	bClamp_AClamped : BOOL := FALSE;
	bClamp_BClamped : BOOL := FALSE;
	
	bAllStop : BOOL;
	
	// For stopping movement & changing modes
	nStopCounter : INT := 0;	// Don't use me.
END_VAR

VAR CONSTANT
	WX2TravelPos 	: sBogieArmPosition := (
						nVertPos 	   := 0,
						nVertTolerance := 5,
						
						nRotPos := -300,
						nRotTolerance := 5,
						
						nClampPos := 15,
						nClampTolerance := 2
						);
						
	WX2LoadPos 	: sBogieArmPosition := (
						nVertPos 	   := 0,
						nVertTolerance := 5,
						
						nRotPos := 0,
						nRotTolerance := 5,
						
						nClampPos := 15,
						nClampTolerance := 2
						);
	WX2UnloadPos 	: sBogieArmPosition := (
						nVertPos 	   := 0,
						nVertTolerance := 5,
						
						nRotPos := 0,
						nRotTolerance := 5,
						
						nClampPos := 15,
						nClampTolerance := 2
						);
	WX2SprayAPos 	: sBogieArmPosition := (
						nVertPos 	   := 200,
						nVertTolerance := 5,
						
						nRotPos := -300,
						nRotTolerance := 5,
						
						nClampPos := 450,
						nClampTolerance := 2
						);
						
	WX2SprayBPos 	: sBogieArmPosition := (
						nVertPos 	   := 200,
						nVertTolerance := 5,
						
						nRotPos := 300,
						nRotTolerance := 5,
						
						nClampPos := 450,
						nClampTolerance := 2
						);
						
	WX2LiftedPos 	: sBogieArmPosition := (
						nVertPos 	   := 200,
						nVertTolerance := 5,
						
						nRotPos := 0,
						nRotTolerance := 5,
						
						nClampPos := 450,
						nClampTolerance := 2
						);
END_VAR

IF WX^.bPresetMoveTrigger THEN
	WX^.bPresetMoveTrigger := FALSE;
END_IF

bAllStop := allAxisAreStopped();

IF bError AND NOT nMoveState = REMOVE_ERROR THEN
	nMoveState := ERROR;
END_IF

IF bCleanUp THEN
	enableAltSpeed();
END_IF

 // WX1^.Vert_A.Out.DistancePos_PO; To get the current location.
IF NOT bInit THEN
	bInit := TRUE;
END_IF

IF GVL_HMI.AutoMode THEN
	CASE nMoveState OF
		STANDBY: // Do Nothing
			IF bBusy AND NOT bError THEN
				nMoveState := STOP_EXTENDED;
				stopAllMovement();
				disableAltSpeed();
				nCounter := 0;
			END_IF
			
			IF bError THEN nMoveState := ERROR; END_IF
			
		LOAD_POSITION: // Load Position -------------------------------------------------------
			
			IF NOT bBusy THEN
				bBusy := TRUE;
				bMoveComplete := FALSE;
				
				WX2TargetPos := WX2LoadPos;

				WX^.VertDisReq_PI 	:= REAL_TO_INT(WX2TargetPos.nVertPos);
				WX^.RotDegReq_PI  	:= REAL_TO_INT(WX2TargetPos.nRotPos);
				WX^.ClampDisReq_PI := 3; // We can assume we are unclamped.
				
				WX^.Clamp_A.bStopMove := FALSE;
				WX^.Clamp_B.bStopMove := FALSE;
				
				startAllMovement();
				
				disableAltSpeed();
				WX^.bPresetMoveTrigger := TRUE;
				
				nMoveState := MAIN_MOVE;
				
				tStartTime := TIME();
				
			ELSE
				nMoveState := STOP;
			END_IF
			
		TRAVERSE_POSITION: // Goto traverse Position -------------------------------------------------------
			
			IF NOT bBusy THEN
				bBusy := TRUE;
				bMoveComplete := FALSE;
				
				WX2TargetPos := WX2TravelPos;

				WX^.VertDisReq_PI 	:= REAL_TO_INT(WX2TargetPos.nVertPos);
				WX^.RotDegReq_PI  	:= REAL_TO_INT(WX2TargetPos.nRotPos);
				WX^.ClampDisReq_PI := REAL_TO_INT(WX^.Clamp_A.Out.DistancePos_PO); // We can assume we are unclamped.
				
				startAllMovement();
				
				disableAltSpeed();
				WX^.bPresetMoveTrigger := TRUE;
				
				nMoveState := MAIN_MOVE;
				
				tStartTime := TIME();
				
			ELSE
				nMoveState := STOP;
			END_IF

		SPRAY_POSITION_A: // Spray Side A -------------------------------------------------------
			IF NOT bBusy THEN
				bBusy := TRUE;
				bMoveComplete := FALSE;
				
				WX2TargetPos := WX2SprayAPos;
				
				WX^.VertDisReq_PI 	:= REAL_TO_INT(WX2TargetPos.nVertPos);
				WX^.RotDegReq_PI  	:= REAL_TO_INT(WX2TargetPos.nRotPos);
				
				WX2TargetPos.nClampPos := WX^.Clamp_A.Out.DistancePos_PO;
				
				startAllMovement();
				disableAltSpeed();
				WX^.bPresetMoveTrigger := TRUE;
				
				nMoveState := MAIN_MOVE;
				
				tStartTime := TIME();
			END_IF
			
		SPRAY_POSITION_B: // Spray Side B -----------------------------------------------------
			IF NOT bBusy THEN
				bBusy := TRUE;
				bMoveComplete := FALSE;
				
				WX2TargetPos := WX2SprayBPos;
				
				WX^.VertDisReq_PI 	:= REAL_TO_INT(WX2TargetPos.nVertPos);
				WX^.RotDegReq_PI  	:= REAL_TO_INT(WX2TargetPos.nRotPos);
				WX2TargetPos.nClampPos := WX^.Clamp_A.Out.DistancePos_PO;
				
				startAllMovement();
				disableAltSpeed();
				WX^.bPresetMoveTrigger := TRUE;
				
				nMoveState := MAIN_MOVE;
				
				tStartTime := TIME();
			END_IF
		
		UNLOAD_POSITION: // Unload Position ||| THIS NEEDS TO BE CHECKED!
			IF NOT bBusy THEN
				bBusy := TRUE;
				bMoveComplete := FALSE;
				
				WX2TargetPos := WX2UnloadPos;
				
				WX^.VertDisReq_PI 	:= REAL_TO_INT(WX2TargetPos.nVertPos);
				WX^.RotDegReq_PI  	:= REAL_TO_INT(WX2TargetPos.nRotPos);
				WX^.ClampDisReq_PI := REAL_TO_INT(WX2TargetPos.nClampPos);
				
				startAllMovement();
				disableAltSpeed();
				WX^.bPresetMoveTrigger := TRUE;
				
				nMoveState := MAIN_MOVE;
				
				tStartTime := TIME();
			END_IF
		
		LIFTED_POSITION:	
			IF NOT bBusy THEN
				bBusy := TRUE;
				bMoveComplete := FALSE;
				
				WX2TargetPos := WX2LiftedPos;
				
				WX^.VertDisReq_PI 	:= REAL_TO_INT(WX2TargetPos.nVertPos);
				WX^.RotDegReq_PI  	:= REAL_TO_INT(WX2TargetPos.nRotPos);
				WX^.ClampDisReq_PI := REAL_TO_INT(WX2TargetPos.nClampPos);
				
				startAllMovement();
				disableAltSpeed();
				WX^.bPresetMoveTrigger := TRUE;
				
				nMoveState := MAIN_MOVE;
				
				tStartTime := TIME();
			END_IF
			
		CLAMP: // Clamp Tool ||||| THIS NEEDS TO BE CHECKED!
			IF NOT bBusy THEN
				bBusy := TRUE;
				bMoveComplete := FALSE;
				
				WX^.ClampDisReq_PI := 500;
				
				tStartTime := TIME();
				
				WX^.Clamp_A.bPresetMoveTrigger := TRUE;
				WX^.Clamp_B.bPresetMoveTrigger := TRUE;
				
				WX^.Clamp_A.bMove_PI := TRUE;
				WX^.Clamp_B.bMove_PI := TRUE;
				
				WX^.Clamp_A.bStopMove := FALSE;
				WX^.Clamp_B.bStopMove := FALSE;
				
				bClamp_AClamped := FALSE;
				bClamp_BClamped := FALSE;
				
					// Set the Clamp Position Tracker to -100, because 0 is a possible clamp value.
				FOR nClampCounter := 1 TO 100 BY 1 DO
					nClamp_ATracker[nClampCounter] := -100;
					nClamp_BTracker[nClampCounter] := -100;
				END_FOR
				nClampCounter := 1;
				disableAltSpeed();
				
				tStartTime := TIME();
			END_IF
			
			
			nClamp_ATracker[nClampCounter] := WX^.Clamp_A.Out.DistancePos_PO;
			nClamp_BTracker[nClampCounter] := WX^.Clamp_B.Out.DistancePos_PO;
			nClampCounter := nClampCounter + 1;
			
				// Checking positions about every 1 second(s)
			IF nClampCounter > 100 THEN
					
				IF TIME() - tStartTime > T#2S THEN
						// Checking Clamp A
					nClampAvgPos := 0;
					IF NOT bClamp_AClamped THEN
						nClampAvgPos := nClamp_ATracker[1];
						
						IF nClampAvgPos = WX^.Clamp_A.Out.DistancePos_PO THEN
							bClamp_AClamped := TRUE;
							nWX2ClampedAPos := WX^.Clamp_A.Out.DistancePos_PO;
						END_IF
					END_IF
					
						// Checking Clamp B
					nClampAvgPos := 0;
					IF NOT bClamp_BClamped THEN
						nClampAvgPos := nClamp_BTracker[1];
						
						IF nClampAvgPos = WX^.Clamp_B.Out.DistancePos_PO THEN
							bClamp_BClamped := TRUE;
							nWX2ClampedBPos := WX^.Clamp_B.Out.DistancePos_PO;
						END_IF
					END_IF
				END_IF
				
				nClampCounter := 1;
			END_IF
				
			IF bClamp_AClamped THEN
				WX^.Clamp_A.bStopMove := TRUE;
			END_IF
			
			IF bClamp_BClamped THEN
				WX^.Clamp_B.bStopMove := TRUE;
			END_IF
			
			IF bClamp_AClamped AND bClamp_BClamped THEN
				IF WX^.Clamp_A.StopCase = 100 AND WX^.Clamp_B.StopCase = 100 THEN
					bClamped   := TRUE;
					WX^.Clamp_A.bStopMove := FALSE;
					WX^.Clamp_B.bStopMove := FALSE;
					nMoveState := STOP;
				END_IF
			END_IF
			
			IF ((TIME() - tStartTime) > tTimeLimit) THEN
				nMoveState := ERROR;
			END_IF
						
			//IF (TIME() - tStartTime) > tTimeLimit THEN
			//	nMoveState := ERROR;
			//	sErrorMessage := 'x Clamping Tool Timeout! x';
			//END_IF
			
		UNCLAMP: // Unclamp Tool ||| THIS NEEDS TO BE CHECKED
			IF NOT bBusy THEN
				bBusy := TRUE;
				bMoveComplete := FALSE;
				
				//WX2^.RotDegReq_PI := LREAL_TO_INT(WX2^.Rot_B.Out.DistancePos_PO);
				WX^.ClampDisReq_PI := 0;
				
				tStartTime := TIME();
				
				WX^.Clamp_A.bPresetMoveTrigger := TRUE;
				WX^.Clamp_B.bPresetMoveTrigger := TRUE;
				
				WX^.Clamp_A.bMove_PI := TRUE;
				WX^.Clamp_B.bMove_PI := TRUE;
				
				WX^.Clamp_A.bStopMove := FALSE;
				WX^.Clamp_B.bStopMove := FALSE;
				
				bClamp_AClamped := TRUE;
				bClamp_BClamped := TRUE;
				
				disableAltSpeed();
				
				bClamped := FALSE;
				
				
				tStartTime := TIME();
			END_IF
			
			IF WX^.Clamp_A.Out.DistancePos_PO < (13) THEN
				WX^.Clamp_A.bStopMove := TRUE;
				bClamp_AClamped := FALSE;
			END_IF
			
			IF WX^.Clamp_B.Out.DistancePos_PO < (13) THEN
				WX^.Clamp_B.bStopMove := TRUE;
				bClamp_BClamped := FALSE;
			END_IF
			IF bClamp_AClamped AND bClamp_BClamped THEN
				bClamped := FALSE;
			END_IF
			
			IF (WX^.Clamp_A.bStopMove AND WX^.Clamp_A.StopCase = 100) AND (WX^.Clamp_B.bStopMove AND WX^.Clamp_B.StopCase = 100) THEN
				nMoveState := STOP;
				WX^.Clamp_A.bStopMove := FALSE;
				WX^.Clamp_B.bStopMove := FALSE;
			END_IF
			
			IF ((TIME() - tStartTime) > tTimeLimit) THEN
				nMoveState := ERROR;
			END_IF
			
		HOME_AXES: // Home each axis
			IF NOT bBusy AND NOT bClamped THEN
				bBusy := TRUE;
				bMoveComplete := FALSE;
				
					// It is 999 to drive the motors into the High Limit Switch for homing off that switch.
				WX^.VertDisReq_PI  := -999;
				WX^.RotDegReq_PI   := -999;
				WX^.ClampDisReq_PI := -999;
				
				WX^.bPresetMoveTrigger := TRUE;
				
				tStartTime := TIME();
			END_IF
			

			IF WX^.Vert_A.bHigh_FI THEN
				WX^.Vert_A.bStopMove := TRUE;
			END_IF
			
			IF WX^.Rot_A.bHigh_FI THEN
				WX^.Rot_A.bStopMove := TRUE;
			END_IF
			
			IF WX^.Clamp_A.bHigh_FI THEN
				WX^.Clamp_A.bStopMove := TRUE;
			END_IF
			
			IF WX^.Vert_B.bHigh_FI THEN
				WX^.Vert_B.bStopMove := TRUE;
			END_IF
			
			IF WX^.Rot_B.bHigh_FI THEN
				WX^.Rot_B.bStopMove := TRUE;
			END_IF
			
			IF WX^.Clamp_B.bHigh_FI THEN
				WX^.Clamp_B.bStopMove := TRUE;
			END_IF
			
			IF WX^.Vert_A.bLow_FI AND WX^.Rot_A.bLow_FI AND WX^.Clamp_A.bLow_FI AND
				WX^.Vert_B.bLow_FI AND WX^.Rot_B.bLow_FI AND WX^.Clamp_B.bLow_FI THEN
				
					WX^.Vert_A.IN.ABSEncoderZero_CI  := WX^.Vert_A.ABSEncoder_FI;//  - (WX2^.Vert_A.IN.SWLimit_Hi_CI  * WX2^.Vert_A.IN.ABSEncoderScaler_CI);
					WX^.Rot_A.IN.ABSEncoderZero_CI   := WX^.Rot_A.ABSEncoder_FI;//   - (WX2^.Rot_A.IN.SWLimit_Hi_CI   * WX2^.Rot_A.IN.ABSEncoderScaler_CI);
					WX^.Clamp_A.IN.ABSEncoderZero_CI := WX^.Clamp_A.ABSEncoder_FI;// - (WX2^.Clamp_A.IN.SWLimit_Hi_CI * WX2^.Clamp_A.IN.ABSEncoderScaler_CI);
					
					WX^.Vert_B.IN.ABSEncoderZero_CI  := WX^.Vert_B.ABSEncoder_FI;//  - (WX2^.Vert_B.IN.SWLimit_Hi_CI  * WX2^.Vert_B.IN.ABSEncoderScaler_CI);
					WX^.Rot_B.IN.ABSEncoderZero_CI   := WX^.Rot_B.ABSEncoder_FI;//   - (WX2^.Rot_B.IN.SWLimit_Hi_CI   * WX2^.Rot_B.IN.ABSEncoderScaler_CI);
					WX^.Clamp_B.IN.ABSEncoderZero_CI := WX^.Clamp_B.ABSEncoder_FI;// - (WX2^.Clamp_B.IN.SWLimit_Hi_CI * WX2^.Clamp_B.IN.ABSEncoderScaler_CI);
					nMoveState := STOP;
			END_IF
			
			IF (TIME() - tStartTime) > tTimeLimit THEN
				nMoveState := ERROR;
				sErrorMessage := 'x Homing Axis Timeout! x';
			END_IF
				
			
		STOP: // Stop All Auto Movement
			disableAltSpeed();
			stopAllMovement();
			bCleanup 			:= FALSE;
			bCleanUpBusy 		:= FALSE;
			bInitCleanupTrigger := FALSE;
			bMoveComplete 		:= TRUE;
			nMoveState 	  		:= STANDBY;
			WX^.bPresetMoveTrigger := FALSE;
			WX^.Vert_A.bPresetMoveTrigger := FALSE;
			WX^.Rot_A.bPresetMoveTrigger := FALSE;
			WX^.Clamp_A.bPresetMoveTrigger := FALSE;
			WX^.Vert_B.bPresetMoveTrigger := FALSE;
			WX^.Rot_B.bPresetMoveTrigger := FALSE;
			WX^.Clamp_B.bPresetMoveTrigger := FALSE;
			
		STOP_EXTENDED:
			IF nStopCounter < 7 THEN
				stopAllMovement();
				disableAltSpeed();
				nStopCounter := nStopCounter + 1;
				
				WX^.bPresetMoveTrigger := FALSE;
				WX^.Vert_A.bPresetMoveTrigger := FALSE;
				WX^.Rot_A.bPresetMoveTrigger := FALSE;
				WX^.Clamp_A.bPresetMoveTrigger := FALSE;
				WX^.Vert_B.bPresetMoveTrigger := FALSE;
				WX^.Rot_B.bPresetMoveTrigger := FALSE;
				WX^.Clamp_B.bPresetMoveTrigger := FALSE;
			ELSE
				stopAllMovement();
				disableAltSpeed();
				nMoveState := STANDBY;
				nStopCounter := 0;
				bBusy := FALSE;
			END_IF
		
		ERROR:
			disableAltSpeed();			
			bError 					:= TRUE;
			bCleanup 				:= FALSE;
			WX^.bPresetMoveTrigger := FALSE;
			stopAllMovement();
			
		REMOVE_ERROR:
			bError 		:= FALSE;
			nMoveState  := STOP;
			
			

			
		CLEAN_UP:
			IF CleanUpMove()THEN				
				nMoveState 			:= CHECK;
				bInitCleanUpTrigger := FALSE;
				nCounter := 0;
			END_IF
			
			IF ((TIME() - tStartTime) > tTimeLimit) THEN
				nMoveState := ERROR;
			END_IF
		
		MAIN_MOVE:
					disableAltSpeed();
			IF armsInTargetPosition() THEN
				bCleanUp := TRUE;
				nMoveState := CLEAN_UP;
				startAllMovement();
			END_IF
			
			IF ((TIME() - tStartTime) > tTimeLimit) THEN
				nMoveState := ERROR;
			END_IF
			
			
			// This is for checking the position to verify that the arms are in the correct position
			// This really is necessary, because we need to throw an error if it is incorrect!
			// Currently just moves to the stop state for testing
		CHECK: 
			(*
			IF NOT precisionMoveChecker() AND bCleanup THEN
				enableAltSpeed();
				IF NOT bClamped THEN
					WX2^.VertDisReq_PI  := LREAL_TO_INT(WX2TargetPos.nVertPos);
					WX2^.RotDegReq_PI 	:= LREAL_TO_INT(WX2TargetPos.nRotPos);
					WX2^.ClampDisReq_PI := LREAL_TO_INT(WX2TargetPos.nClampPos);
					
					WX2^.bPresetMoveTrigger := TRUE;
				ELSE
					WX2^.VertDisReq_PI  := LREAL_TO_INT(WX2TargetPos.nVertPos);
					WX2^.RotDegReq_PI 	:= LREAL_TO_INT(WX2TargetPos.nRotPos);
					
					WX2^.Vert_A.bMove_PI := TRUE;
					WX2^.Vert_A.bPresetMoveTrigger := TRUE;
					
					WX2^.Vert_B.bMove_PI := TRUE;
					WX2^.Vert_B.bPresetMoveTrigger := TRUE;
					
					WX2^.Rot_A.bMove_PI := TRUE;
					WX2^.Rot_A.bPresetMoveTrigger := TRUE;
				END_IF
			ELSE
				nMoveState := STOP;
			END_IF
			*)
			nMoveState := STOP;
	END_CASE
	
		// If holding tool, then we disable the clamp and follow rotation axis
	IF bClamped THEN
				// If we are clamped and NOT unloading, then we disable the follow rotation axis,
				// 		otherwise we need that axis enabled to put the tool down safely.
		WX^.Rot_B.EnableOut_FO := FALSE;
		WX^.Rot_B.bStopMove := TRUE;
		WX^.Clamp_A.EnableOut_FO := FALSE;
		WX^.Clamp_B.EnableOut_FO := FALSE;
		WX^.Clamp_A.bStopMove := TRUE;
		WX^.Clamp_B.bStopMove := TRUE;
		
		 // Unclamping detection.
		 (* This uses the scaled encoder value. Maybe should be changed to absolute encoder value. *)
		IF (nWX2ClampedAPos > (nClampTolerance + WX^.Clamp_A.Out.DistancePos_PO)) THEN
			bError := TRUE;
			sErrorMessage := 'A side clamp has become unlclamped!';
		END_IF
		IF (nWX2ClampedBPos > (nClampTolerance + WX^.Clamp_B.Out.DistancePos_PO)) THEN
			bError := TRUE;
			sErrorMessage := 'B side clamp has become unlclamped!';
		END_IF
	ELSE
		IF (NOT nMoveState = UNCLAMP) THEN
			WX^.Clamp_A.bPresetMoveTrigger := FALSE;
			WX^.Clamp_B.bPresetMoveTrigger := FALSE;
		END_IF
	END_IF
END_IF

METHOD allAxisAreStopped : BOOL
VAR
	bVertA 	: BOOL := FALSE;
	bRotA  	: BOOL := FALSE;
	bClampA : BOOL := FALSE;
	bVertB 	: BOOL := FALSE;
	bRotB  	: BOOL := FALSE;
	bClampB : BOOL := FALSE;
END_VAR
IF WX^.Vert_B.StopCase = 100 THEN
	bVertB := TRUE;
END_IF

IF WX^.Rot_B.StopCase = 100 THEN
	bRotB := TRUE;
END_IF

IF WX^.Clamp_B.StopCase = 100 THEN
	bClampB := TRUE;
END_IF

IF WX^.Vert_A.StopCase = 100 THEN
	bVertA := TRUE;
END_IF

IF WX^.Rot_A.StopCase = 100 THEN
	bRotA := TRUE;
END_IF

IF WX^.Clamp_A.StopCase = 100 THEN
	bClampA := TRUE;
END_IF

allAxisAreStopped := bVertA AND bRotA AND bClampA AND bVertB AND bRotB AND bClampB;
END_METHOD

METHOD armsInTargetPosition : BOOL
VAR	
	bInPosition : BOOL := FALSE;
END_VAR
//WX1

//WX2
	// WX2A VERT
IF WX2TargetPos.nVertPos + WX2TargetPos.nVertCatch > WX^.Vert_A.Out.DistancePos_PO AND
	WX2TargetPos.nVertPos - WX2TargetPos.nVertCatch < WX^.Vert_A.Out.DistancePos_PO THEN
		WX^.Vert_A.bStopMove := TRUE;
END_IF

